// TIA Portal V18 program export: 5 tag tables, 0 data types, 1 data blocks, 15 code blocks (in call order from the OBs), 44 instance data blocks

VAR_GLOBAL   // PLC tag table "AI"
   "H/SSR_019_TT01_IN" AT %IW70 : Int;
   "H/SSR_019_TT02_IN" AT %IW72 : Int;
   "H/SSR_019_APT01_IN" AT %IW74 : Int;
   "H/SSR_019_GPT101_IN" AT %IW78 : Int;
   "H/SSR_019_GPT201_IN" AT %IW80 : Int;
   "H/SSR_019_GPT301_IN" AT %IW82 : Int;
   "H/SSR_019_GPT401_IN" AT %IW84 : Int;
   "H/SSR_019_GPT501_IN" AT %IW86 : Int;
   "H/SSR_019_GPT601_IN" AT %IW88 : Int;
   "H/SSR_019_TT03_IN" AT %IW76 : Int;
   Tag_1 AT %T5 : Timer;
END_VAR

VAR_GLOBAL   // PLC tag table "AO"
   "H/SSR_019_CV01_CVOUT" AT %QW26 : Int;
   "H/SSR_019_CV02_CVOUT" AT %QW28 : Int;
   "H/SSR_019_CV03_CVOUT" AT %QW30 : Int;
   SPARE AT %QW38 : Int;
   SPARE_1 AT %QW40 : Int;
   SPARE_2 AT %QW42 : Int;
   SPARE_3 AT %QW44 : Int;
   SPARE_4 AT %QW46 : Int;
   SPARE_5 AT %QW48 : Int;
   SPARE_6 AT %QW50 : Int;
   SPARE_7 AT %QW52 : Int;
   SPARE_8 AT %QW54 : Int;
   SPARE_9 AT %QW56 : Int;
   SPARE_10 AT %QW58 : Int;
   SPARE_11 AT %QW60 : Int;
   SPARE_12 AT %QW62 : Int;
   SPARE_13 AT %QW64 : Int;
   SPARE_14 AT %QW66 : Int;
END_VAR

VAR_GLOBAL   // PLC tag table "DI"
   "H/SSR_019_XV01_OPENFB" AT %I7.4 : Bool;
   "H/SSR_019_XV01_CLOSEFB" AT %I7.5 : Bool;
   "H/SSR_019_XV02_OPENFB" AT %I7.6 : Bool;
   "H/SSR_019_XV02_CLOSEFB" AT %I7.7 : Bool;
   "H/SSR_019_XV03_OPENFB" AT %I8.0 : Bool;
   "H/SSR_019_XV03_CLOSEFB" AT %I8.1 : Bool;
   "H/SSR_019_XV04_CLOSEFB" AT %I8.2 : Bool;
   "H/SSR_019_XV04_OPENFB" AT %I8.3 : Bool;
   "H/SSR_019_XV05_OPENFB" AT %I8.4 : Bool;
   "H/SSR_019_XV05_CLOSEFB" AT %I8.5 : Bool;
   "H/SSR_019_XV06_OPENFB" AT %I8.6 : Bool;
   "H/SSR_019_XV06_CLOSEFB" AT %I8.7 : Bool;
   "H/SSR_019_XV07_OPENFB" AT %I9.0 : Bool;
   "H/SSR_019_XV07_CLOSEFB" AT %I9.1 : Bool;
   "H/SSR_019_XV08_OPENFB" AT %I9.2 : Bool;
   "H/SSR_019_XV08_CLOSEFB" AT %I9.3 : Bool;
   "H/SSR_019_XV09_OPENFB" AT %I9.4 : Bool;
   "H/SSR_019_XV09_CLOSEFB" AT %I9.5 : Bool;
   "H/SSR_019_XV10_OPENFB" AT %I9.6 : Bool;
   "H/SSR_019_XV10_CLOSEFB" AT %I9.7 : Bool;
   "H/SSR_019_XV11_OPENFB" AT %I10.0 : Bool;
   "H/SSR_019_XV11_CLOSEFB" AT %I10.1 : Bool;
   "H/SSR_019_XV12_OPENFB" AT %I10.2 : Bool;
   "H/SSR_019_XV12_CLOSEFB" AT %I10.3 : Bool;
   "H/SSR_019_XV13_OPENFB" AT %I10.4 : Bool;
   "H/SSR_019_XV13_CLOSEFB" AT %I10.5 : Bool;
   "H/SSR_019_AG_RUNFB" AT %I10.6 : Bool;
   "H/SSR_019_AG_STOPFB" AT %I10.7 : Bool;
   "H/SSR_019_AG_TRIP" AT %I11.0 : Bool;
END_VAR

VAR_GLOBAL   // PLC tag table "DO"
   "H/SSR_006_XV01_OPEN" AT %Q0.0 : Bool;
   "H/SSR_006_XV02_OPEN" AT %Q0.1 : Bool;
   "H/SSR_006_XV03_OPEN" AT %Q0.2 : Bool;
   "H/SSR_006_XV04_OPEN" AT %Q0.3 : Bool;
   "H/SSR_006_XV05_OPEN" AT %Q0.4 : Bool;
   "H/SSR_006_XV06_OPEN" AT %Q0.5 : Bool;
   "H/SSR_006_XV07_OPEN" AT %Q0.6 : Bool;
   "H/SSR_006_XV08_OPEN" AT %Q0.7 : Bool;
   "H/SSR_006_XV09_OPEN" AT %Q1.0 : Bool;
   "H/SSR_006_XV10_OPEN" AT %Q1.1 : Bool;
   "H/SSR_006_XV11_OPEN" AT %Q1.2 : Bool;
   "H/SSR_006_XV12_OPEN" AT %Q1.3 : Bool;
   "H/SSR_006_XV13_OPEN" AT %Q1.4 : Bool;
   "H/SSR_006_XV14_OPEN" AT %Q1.5 : Bool;
   "H/SSR_006_AG_RUN" AT %Q1.6 : Bool;
   "H/SSR_010_XV01_OPEN" AT %Q1.7 : Bool;
   "H/SSR_010_XV02_OPEN" AT %Q2.0 : Bool;
   "H/SSR_010_XV03_OPEN" AT %Q2.1 : Bool;
   "H/SSR_010_XV04_OPEN" AT %Q2.2 : Bool;
   "H/SSR_010_XV05_OPEN" AT %Q2.3 : Bool;
   "H/SSR_010_XV06_OPEN" AT %Q2.4 : Bool;
   "H/SSR_010_XV07_OPEN" AT %Q2.5 : Bool;
   "H/SSR_010_XV08_OPEN" AT %Q2.6 : Bool;
   "H/SSR_010_XV09_OPEN" AT %Q2.7 : Bool;
   "H/SSR_010_XV10_OPEN" AT %Q3.0 : Bool;
   "H/SSR_010_XV11_OPEN" AT %Q3.1 : Bool;
   "H/SSR_010_XV12_OPEN" AT %Q3.2 : Bool;
   "H/SSR_010_XV13_OPEN" AT %Q3.3 : Bool;
   "H/SSR_010_XV14_OPEN" AT %Q3.4 : Bool;
   "H/SSR_010_AG_RUN" AT %Q3.5 : Bool;
   "H/SSR_019_XV01_OPEN" AT %Q3.6 : Bool;
   "H/SSR_019_XV02_OPEN" AT %Q3.7 : Bool;
   "H/SSR_019_XV03_OPEN" AT %Q4.0 : Bool;
   "H/SSR_019_XV04_OPEN" AT %Q4.1 : Bool;
   "H/SSR_019_XV05_OPEN" AT %Q4.2 : Bool;
   "H/SSR_019_XV06_OPEN" AT %Q4.3 : Bool;
   "H/SSR_019_XV07_OPEN" AT %Q4.4 : Bool;
   "H/SSR_019_XV08_OPEN" AT %Q4.5 : Bool;
   "H/SSR_019_XV09_OPEN" AT %Q4.6 : Bool;
   "H/SSR_019_XV10_OPEN" AT %Q4.7 : Bool;
   "H/SSR_019_XV11_OPEN" AT %Q5.0 : Bool;
   "H/SSR_019_XV12_OPEN" AT %Q5.1 : Bool;
   "H/SSR_019_XV13_OPEN" AT %Q5.2 : Bool;
   "H/SSR_019_XV14_OPEN" AT %Q5.3 : Bool;
   "H/SSR_019_AG_RUN" AT %Q5.4 : Bool;
   "H/SSR_020_XV01_OPEN" AT %Q5.5 : Bool;
   "H/SSR_020_XV02_OPEN" AT %Q5.6 : Bool;
   "H/SSR_020_XV03_OPEN" AT %Q5.7 : Bool;
   "H/SSR_020_XV04_OPEN" AT %Q6.0 : Bool;
   "H/SSR_020_XV05_OPEN" AT %Q6.1 : Bool;
   "H/SSR_020_XV06_OPEN" AT %Q6.2 : Bool;
   "H/SSR_020_XV07_OPEN" AT %Q6.3 : Bool;
   "H/SSR_020_XV08_OPEN" AT %Q6.4 : Bool;
   "H/SSR_020_XV09_OPEN" AT %Q6.5 : Bool;
   "H/SSR_020_XV10_OPEN" AT %Q6.6 : Bool;
   "H/SSR_020_XV11_OPEN" AT %Q6.7 : Bool;
   "H/SSR_020_XV12_OPEN" AT %Q7.0 : Bool;
   "H/SSR_020_XV13_OPEN" AT %Q7.1 : Bool;
   "H/SSR_020_XV14_OPEN" AT %Q7.2 : Bool;
   "H/SSR_020_AG_RUN" AT %Q7.3 : Bool;
   DO_SPARE_1 AT %Q7.4 : Bool;
   DO_SPARE_2 AT %Q7.5 : Bool;
   DO_SPARE_3 AT %Q7.6 : Bool;
   DO_SPARE_4 AT %Q7.7 : Bool;
   DO_SPARE_5 AT %Q8.0 : Bool;
   DO_SPARE_6 AT %Q8.1 : Bool;
   DO_SPARE_7 AT %Q8.2 : Bool;
   DO_SPARE_8 AT %Q8.3 : Bool;
   DO_SPARE_9 AT %Q8.4 : Bool;
   DO_SPARE_10 AT %Q8.5 : Bool;
   DO_SPARE_11 AT %Q8.6 : Bool;
   DO_SPARE_12 AT %Q8.7 : Bool;
   DO_SPARE_13 AT %Q9.0 : Bool;
   DO_SPARE_14 AT %Q9.1 : Bool;
   DO_SPARE_15 AT %Q9.2 : Bool;
   DO_SPARE_16 AT %Q9.3 : Bool;
   DO_SPARE_17 AT %Q9.4 : Bool;
   DO_SPARE_18 AT %Q9.5 : Bool;
   DO_SPARE_19 AT %Q9.6 : Bool;
   DO_SPARE_20 AT %Q9.7 : Bool;
   DO_SPARE_21 AT %Q10.0 : Bool;
   DO_SPARE_22 AT %Q10.1 : Bool;
   DO_SPARE_23 AT %Q10.2 : Bool;
   DO_SPARE_24 AT %Q10.3 : Bool;
   DO_SPARE_25 AT %Q10.4 : Bool;
   DO_SPARE_26 AT %Q10.5 : Bool;
   DO_SPARE_27 AT %Q10.6 : Bool;
   DO_SPARE_28 AT %Q10.7 : Bool;
   DO_SPARE_29 AT %Q11.0 : Bool;
   DO_SPARE_30 AT %Q11.1 : Bool;
   DO_SPARE_31 AT %Q11.2 : Bool;
   DO_SPARE_32 AT %Q11.3 : Bool;
   DO_SPARE_33 AT %Q11.4 : Bool;
   DO_SPARE_34 AT %Q11.5 : Bool;
   DO_SPARE_35 AT %Q11.6 : Bool;
   DO_SPARE_36 AT %Q11.7 : Bool;
   DO_SPARE_37 AT %Q12.0 : Bool;
   DO_SPARE_38 AT %Q12.1 : Bool;
   DO_SPARE_39 AT %Q12.2 : Bool;
   DO_SPARE_40 AT %Q12.3 : Bool;
   DO_SPARE_41 AT %Q12.4 : Bool;
   DO_SPARE_42 AT %Q12.5 : Bool;
   DO_SPARE_43 AT %Q12.6 : Bool;
   DO_SPARE_44 AT %Q12.7 : Bool;
   DO_SPARE_45 AT %Q13.0 : Bool;
   DO_SPARE_46 AT %Q13.1 : Bool;
   DO_SPARE_47 AT %Q13.2 : Bool;
   DO_SPARE_48 AT %Q13.3 : Bool;
   DO_SPARE_49 AT %Q13.4 : Bool;
   DO_SPARE_50 AT %Q13.5 : Bool;
   DO_SPARE_51 AT %Q13.6 : Bool;
   DO_SPARE_52 AT %Q13.7 : Bool;
END_VAR

VAR_GLOBAL   // PLC tag table "Default tag table_1"
   System_Byte AT %MB1 : Byte;
   FirstScan AT %M1.0 : Bool;
   DiagStatusUpdate AT %M1.1 : Bool;
   AlwaysTRUE AT %M1.2 : Bool;
   AlwaysFALSE AT %M1.3 : Bool;
   Clock_Byte AT %MB0 : Byte;
   Clock_10Hz AT %M0.0 : Bool;
   Clock_5Hz AT %M0.1 : Bool;
   "Clock_2.5Hz" AT %M0.2 : Bool;
   Clock_2Hz AT %M0.3 : Bool;
   "Clock_1.25Hz" AT %M0.4 : Bool;
   Clock_1Hz AT %M0.5 : Bool;
   "Clock_0.625Hz" AT %M0.6 : Bool;
   "Clock_0.5Hz" AT %M0.7 : Bool;
   "H/SSR_019_START" AT %M2.0 : Bool;
   "H/SSR_019_SP" AT %MD4 : Real;
   "H/SSR_019_TT01_PV" AT %MD8 : Real;
   "H/SSR_019_ALERT_SP" AT %MD12 : Real;
   "H/SSR_019_CHBr_RT_SP" AT %MD16 : Real;
   "H/SSR_019_RT_HW_SP" AT %MD20 : Real;
   "H/SSR_019_HW_STEAM_SP" AT %MD24 : Real;
   "H/SSR_019_RT_CHBr_SP" AT %MD28 : Real;
   "H/SSR_019_SOURCE_SEL" AT %MW32 : Int;
   "H/SSR_019_AM" AT %M2.1 : Bool;
   "H/SSR_019_TIME_SP" AT %MW34 : Int;
   "H/SSR_019_KP" AT %MW36 : Int;
   "H/SSR_019_TI" AT %MW38 : Int;
   "H/SSR_019_TT02_PV" AT %MD40 : Real;
   "H/SSR_019_CV02_MANOUT" AT %MD44 : Real;
   "H/SSR_019_START_PV" AT %MD48 : Real;
   "H/SSR_019_CV02_SCVOUT" AT %MD52 : Real;
   "H/SSR_019_RUN_MIN" AT %MW56 : Int;
   "H/SSR_019_FLUSH_TIME_SP" AT %MW60 : Int;
   "H/SSR_019_VENT_TIME_SP" AT %MW62 : Int;
   "H/SSR_019_CONDENSATE_TIME_SP" AT %MW64 : Int;
   "H/SSR_019_XV01_CMD" AT %M58.7 : Bool;
   "H/SSR_019_XV02_CMD" AT %M59.0 : Bool;
   "H/SSR_019_XV03_CMD" AT %M59.1 : Bool;
   "H/SSR_019_XV07_CMD" AT %M59.2 : Bool;
   "H/SSR_019_XV08_CMD" AT %M59.3 : Bool;
   "H/SSR_019_XV09_CMD" AT %M59.4 : Bool;
   "H/SSR_019_XV11_CMD" AT %M59.5 : Bool;
   "H/SSR_019_XV12_CMD" AT %M59.6 : Bool;
   "H/SSR_019_XV13_CMD" AT %M59.7 : Bool;
   "H/SSR_019_XV10_CMD" AT %M66.0 : Bool;
   "H/SSR_019_XV05_CMD" AT %M66.1 : Bool;
   "H/SSR_019_XV06_CMD" AT %M66.2 : Bool;
   "H/SSR_019_FLUSH_RUN_TIME" AT %MD68 : Real;
   "H/SSR_019_CONDENSATE_RUN_TIME" AT %MD72 : Real;
   "H/SSR_019_VENT_RUN_TIME" AT %MD76 : Real;
   "H/SSR_019_CV01_MANOUT" AT %MD80 : Real;
   "H/SSR_019_CV01_SCVOUT" AT %MD84 : Real;
   "H/SSR_019_HOLD" AT %M66.3 : Bool;
   "H/SSR_019_EMSTOP" AT %M66.4 : Bool;
   XV_ERRORMON_TIME AT %MD88 : Time;
   "H/SSR_019_XV01_RESET" AT %M66.5 : Bool;
   "H/SSR_019_XV01_MCMD" AT %M66.6 : Bool;
   "H/SSR_019_XV01_Status" AT %MW92 : Word;
   "H/SSR_019_XV02_MCMD" AT %M66.7 : Bool;
   "H/SSR_019_XV02_RESET" AT %M67.0 : Bool;
   "H/SSR_019_XV03_MCMD" AT %M67.1 : Bool;
   "H/SSR_019_XV03_RESET" AT %M67.2 : Bool;
   "H/SSR_019_XV04_MCMD" AT %M67.3 : Bool;
   "H/SSR_019_XV04_RESET" AT %M67.4 : Bool;
   "H/SSR_019_XV05_MCMD" AT %M67.5 : Bool;
   "H/SSR_019_XV05_RESET" AT %M67.6 : Bool;
   "H/SSR_019_XV06_MCMD" AT %M67.7 : Bool;
   "H/SSR_019_XV06_RESET" AT %M94.0 : Bool;
   "H/SSR_019_XV07_MCMD" AT %M94.1 : Bool;
   "H/SSR_019_XV07_RESET" AT %M94.2 : Bool;
   "H/SSR_019_XV08_MCMD" AT %M94.3 : Bool;
   "H/SSR_019_XV08_RESET" AT %M94.4 : Bool;
   "H/SSR_019_XV09_MCMD" AT %M94.5 : Bool;
   "H/SSR_019_XV09_RESET" AT %M94.6 : Bool;
   "H/SSR_019_XV10_MCMD" AT %M94.7 : Bool;
   "H/SSR_019_XV10_RESET" AT %M95.0 : Bool;
   "H/SSR_019_XV11_MCMD" AT %M95.1 : Bool;
   "H/SSR_019_XV11_RESET" AT %M95.2 : Bool;
   "H/SSR_019_XV12_MCMD" AT %M95.3 : Bool;
   "H/SSR_019_XV12_RESET" AT %M95.4 : Bool;
   "H/SSR_019_XV13_MCMD" AT %M95.5 : Bool;
   "H/SSR_019_XV13_RESET" AT %M95.6 : Bool;
   "H/SSR_019_XV02_Status" AT %MW96 : Word;
   "H/SSR_019_XV03_Status" AT %MW98 : Word;
   "H/SSR_019_XV04_Status" AT %MW100 : Word;
   "H/SSR_019_XV05_Status" AT %MW102 : Word;
   "H/SSR_019_XV07_Status" AT %MW104 : Word;
   "H/SSR_019_XV08_Status" AT %MW106 : Word;
   "H/SSR_019_XV09_Status" AT %MW108 : Word;
   "H/SSR_019_XV10_Status" AT %MW110 : Word;
   "H/SSR_019_XV06_Status" AT %MW112 : Word;
   "H/SSR_019_XV11_Status" AT %MW114 : Word;
   "H/SSR_019_XV12_Status" AT %MW116 : Word;
   "H/SSR_019_XV13_Status" AT %MW118 : Word;
   "H/SSR_019_CV03_SCVOUT" AT %MW120 : Int;
   "H/SSR_019_APT01_PV" AT %MD122 : Real;
   "H/SSR_019_AG_CMD" AT %M2.2 : Bool;
   "H/SSR_019_AG_MCMD" AT %M2.3 : Bool;
   "H/SSR_019_AG_RESET" AT %M2.4 : Bool;
   "H/SSR_019_AG_Status" AT %MW126 : Word;
   "H/SSR_019_CV03_MANOUT" AT %MD128 : Real;
   "H/SSR_019_TT01_Faulty" AT %M2.5 : Bool;
   "H/SSR_019_APT01_Faulty" AT %M2.6 : Bool;
   "H/SSR_019_TT02_Faulty" AT %M2.7 : Bool;
   "H/SSR_019_TT01_Fault" AT %M3.0 : Bool;
   "H/SSR_019_ALERT_SP_EMPTY" AT %M3.1 : Bool;
   "H/SSR_019_SP_EMPTY" AT %M3.2 : Bool;
   "H/SSR_019_CHANGEOVER_SP_EMPTY" AT %M3.3 : Bool;
   "H/SSR_019_FlushTime_SP_EMPTY" AT %M3.4 : Bool;
   "H/SSR_019_VentTime_SP_EMPTY" AT %M3.5 : Bool;
   "H/SSR_019_Cond_Time_EMPTY" AT %M3.6 : Bool;
   "H/SSR_019_XV01_Faulty" AT %M3.7 : Bool;
   "H/SSR_019_XV02_Faulty" AT %M58.0 : Bool;
   "H/SSR_019_XV03_Faulty" AT %M58.1 : Bool;
   "H/SSR_019_XV04_Faulty" AT %M58.2 : Bool;
   "H/SSR_019_XV05_Faulty" AT %M58.3 : Bool;
   "H/SSR_019_XV06_Faulty" AT %M58.4 : Bool;
   "H/SSR_019_XV07_Faulty" AT %M58.5 : Bool;
   "H/SSR_019_XV08_Faulty" AT %M58.6 : Bool;
   "H/SSR_019_XV09_Faulty" AT %M95.7 : Bool;
   "H/SSR_019_XV10_Faulty" AT %M132.0 : Bool;
   "H/SSR_019_XV11_Faulty" AT %M132.1 : Bool;
   "H/SSR_019_XV12_Faulty" AT %M132.2 : Bool;
   "H/SSR_019_XV13_Faulty" AT %M132.3 : Bool;
   "H/SSR_019_Flush_CMP" AT %M132.4 : Bool;
   "H/SSR_019_Vent_CMP" AT %M132.5 : Bool;
   "H/SSR_019_Cond_CMP" AT %M134.0 : Bool;
   "H/SSR_019_GPT101_Fault" AT %M134.1 : Bool;
   "H/SSR_019_GPT101_PV" AT %MD130 : Real;
   "H/SSR_019_GPT201_PV" AT %MD134 : Real;
   "H/SSR_019_GPT201_Fault" AT %M134.2 : Bool;
   "H/SSR_019_GPT301_Fault" AT %M134.3 : Bool;
   "H/SSR_019_GPT401_Fault" AT %M134.4 : Bool;
   "H/SSR_019_GPT501_Fault" AT %M134.5 : Bool;
   "H/SSR_019_GPT601_Fault" AT %M134.6 : Bool;
   "H/SSR_019_TT03_Fault" AT %M135.0 : Bool;
   "H/SSR_019_GPT301_PV" AT %MD132 : Real;
   "H/SSR_019_GPT401_PV" AT %MD135 : Real;
   "H/SSR_019_GPT501_PV" AT %MD136 : Real;
   "H/SSR_019_GPT601_PV" AT %MD137 : Real;
   "H/SSR_019_RESET" AT %M134.7 : Bool;
   "H/SSR_019_TT103_PV" AT %MD138 : Real;
   "H/SSR_019_HOOTER_Status" AT %M135.1 : Bool;
END_VAR
VAR_GLOBAL CONSTANT   // user constants
   "None(1)" : Pip := 65535;
   "Automatic update(1)" : Pip := 0;
   "PIP 1(1)" : Pip := 1;
   "PIP 2(1)" : Pip := 2;
   "PIP 3(1)" : Pip := 3;
   "PIP 4(1)" : Pip := 4;
   "PIP 5(1)" : Pip := 5;
   "PIP 6(1)" : Pip := 6;
   "PIP 7(1)" : Pip := 7;
   "PIP 8(1)" : Pip := 8;
   "PIP 9(1)" : Pip := 9;
   "PIP 10(1)" : Pip := 10;
   "PIP 11(1)" : Pip := 11;
   "PIP 12(1)" : Pip := 12;
   "PIP 13(1)" : Pip := 13;
   "PIP 14(1)" : Pip := 14;
   "PIP 15(1)" : Pip := 15;
   "PIP 16(1)" : Pip := 16;
   "PIP 17(1)" : Pip := 17;
   "PIP 18(1)" : Pip := 18;
   "PIP 19(1)" : Pip := 19;
   "PIP 20(1)" : Pip := 20;
   "PIP 21(1)" : Pip := 21;
   "PIP 22(1)" : Pip := 22;
   "PIP 23(1)" : Pip := 23;
   "PIP 24(1)" : Pip := 24;
   "PIP 25(1)" : Pip := 25;
   "PIP 26(1)" : Pip := 26;
   "PIP 27(1)" : Pip := 27;
   "PIP 28(1)" : Pip := 28;
   "PIP 29(1)" : Pip := 29;
   "PIP 30(1)" : Pip := 30;
   "PIP 31(1)" : Pip := 31;
   "Local1~MC" : Hw_SubModule := 65151;
   "Local1~Common" : Hw_SubModule := 65150;
   "Local1~Device" : Hw_Device := 65132;
   "Local1~Configuration" : Hw_SubModule := 65133;
   "Local1~RHSystem" : Hw_Device := 34;
   "Local1~Display" : Hw_SubModule := 65154;
   "Local1~Exec" : Hw_SubModule := 65152;
   Local1 : Hw_SubModule := 65149;
   "Local1~PROFINET_interface_1" : Hw_Interface := 65164;
   "Local1~PROFINET_interface_1~Port_1" : Hw_Interface := 65165;
   "Local1~PROFINET_interface_1~Port_2" : Hw_Interface := 65166;
   "Local1~PROFINET_interface_1~HsystemIPRef_1" : Hw_Interface := 257;
   "Local1~HCPUredCtrl" : Hw_SubModule := 65147;
   "Local2~MC" : Hw_SubModule := 65351;
   "Local2~Common" : Hw_SubModule := 65350;
   "Local2~Device" : Hw_Device := 65332;
   "Local2~Configuration" : Hw_SubModule := 65333;
   "Local2~Display" : Hw_SubModule := 65354;
   "Local2~Exec" : Hw_SubModule := 65352;
   Local2 : Hw_SubModule := 65349;
   "Local2~PROFINET_interface_1" : Hw_Interface := 65364;
   "Local2~PROFINET_interface_1~Port_1" : Hw_Interface := 65365;
   "Local2~PROFINET_interface_1~Port_2" : Hw_Interface := 65366;
   "Local2~PROFINET_interface_1~HsystemIPRef_1" : Hw_Interface := 268;
   "Local2~HCPUredCtrl" : Hw_SubModule := 65347;
   "OB_AutoLogic(1)" : OB_PCYCLE := 1;
   "OB_Main(1)" : OB_PCYCLE := 123;
   "OB_PID Cyclic interrupt(1)" : OB_Cyclic := 30;
   "OB_Cyclic interrupt(1)" : OB_Cyclic := 31;
END_VAR

DATA_BLOCK "SIM_VALVE"   // DB29
{ S7_Optimized_Access := 'FALSE' }
VERSION : 0.1
// stored: AutoNumber true, DBAccessibleFromOPCUA true, DBAccessibleFromWebserver true, IsOnlyStoredInLoadMemory false, IsWriteProtectedInAS false
   VAR
      "H/SSR_019_XV01_CLOSEFB" : Bool;
      "H/SSR_019_XV02_OPENFB" : Bool;
      "H/SSR_019_XV02_CLOSEFB" : Bool;
      "H/SSR_019_XV03_OPENFB" : Bool;
      "H/SSR_019_XV03_CLOSEFB" : Bool;
      "H/SSR_019_XV04_CLOSEFB" : Bool;
      "H/SSR_019_XV04_OPENFB" : Bool;
      "H/SSR_019_XV05_OPENFB" : Bool;
      "H/SSR_019_XV05_CLOSEFB" : Bool;
      "H/SSR_019_XV06_OPENFB" : Bool;
      "H/SSR_019_XV06_CLOSEFB" : Bool;
      "H/SSR_019_XV07_OPENFB" : Bool;
      "H/SSR_019_XV07_CLOSEFB" : Bool;
      "H/SSR_019_XV08_OPENFB" : Bool;
      "H/SSR_019_XV08_CLOSEFB" : Bool;
      "H/SSR_019_XV09_OPENFB" : Bool;
      "H/SSR_019_XV09_CLOSEFB" : Bool;
      "H/SSR_019_XV10_OPENFB" : Bool;
      "H/SSR_019_XV10_CLOSEFB" : Bool;
      "H/SSR_019_XV11_OPENFB" : Bool;
      "H/SSR_019_XV11_CLOSEFB" : Bool;
      "H/SSR_019_XV12_OPENFB" : Bool;
      "H/SSR_019_XV12_CLOSEFB" : Bool;
      "H/SSR_019_XV13_OPENFB" : Bool;
      "H/SSR_019_XV13_CLOSEFB" : Bool;
      "H/SSR_019_TT01_IN" : Int;
      "H/SSR_019_TT02_IN" : Int;
      "H/SSR_019_APT01_IN" : Int;
      "H/SSR_019_GPT101_IN" : Int;
      "H/SSR_019_GPT201_IN" : Int;
      "H/SSR_019_GPT301_IN" : Int;
      "H/SSR_019_GPT401_IN" : Int;
      "H/SSR_019_GPT501_IN" : Int;
      "H/SSR_019_GPT601_IN" : Int;
      "H/SSR_019_TT03_IN" : Int;
      "H/SSR_019_TT01_PV" : Int;
      "H/SSR_019_XV01_OPENFB" : Bool;
      "H/SSR_019_TT02_INpv" : Bool;
      "H/SSR_019_APT01_PV" : Bool;
      "H/SSR_019_GPT101_PV" : Bool;
      "H/SSR_019_GPT201_PV" : Bool;
      "H/SSR_019_GPT301_PV" : Bool;
      "H/SSR_019_GPT401_PV" : Bool;
      "H/SSR_019_GPT501_PV" : Bool;
      "H/SSR_019_GPT601_PV" : Bool;
      "H/SSR_019_TT03_PV" : Bool;
      "H/SSR_019_TT01_PV_1" : Bool;
   END_VAR
BEGIN
END_DATA_BLOCK

ORGANIZATION_BLOCK "AutoLogic"   // OB1, FBD, ProgramCycle
TITLE = "Main Program Sweep (Cycle)"
{ S7_Optimized_Access := 'TRUE' }
VERSION : 0.1
// stored: AutoNumber true, IsIECCheckEnabled false, SetENOAutomatically false
   VAR_INPUT
      Initial_Call : Bool;   // Initial call of this OB
      Remanence : Bool;   // =True, if remanent data are available
   END_VAR
   VAR_TEMP
      UTL_TIME : Array[0..2] of DInt;
      chbs_cmd : Bool;
      chbr_cmd : Bool;
      STEAM_MAN_SCV_MVE : Real;
      STEAM_SCV_MVE : Real;
      STEAM_SCV_SCL : Real;
   END_VAR
BEGIN

REGION Network 1: Source select
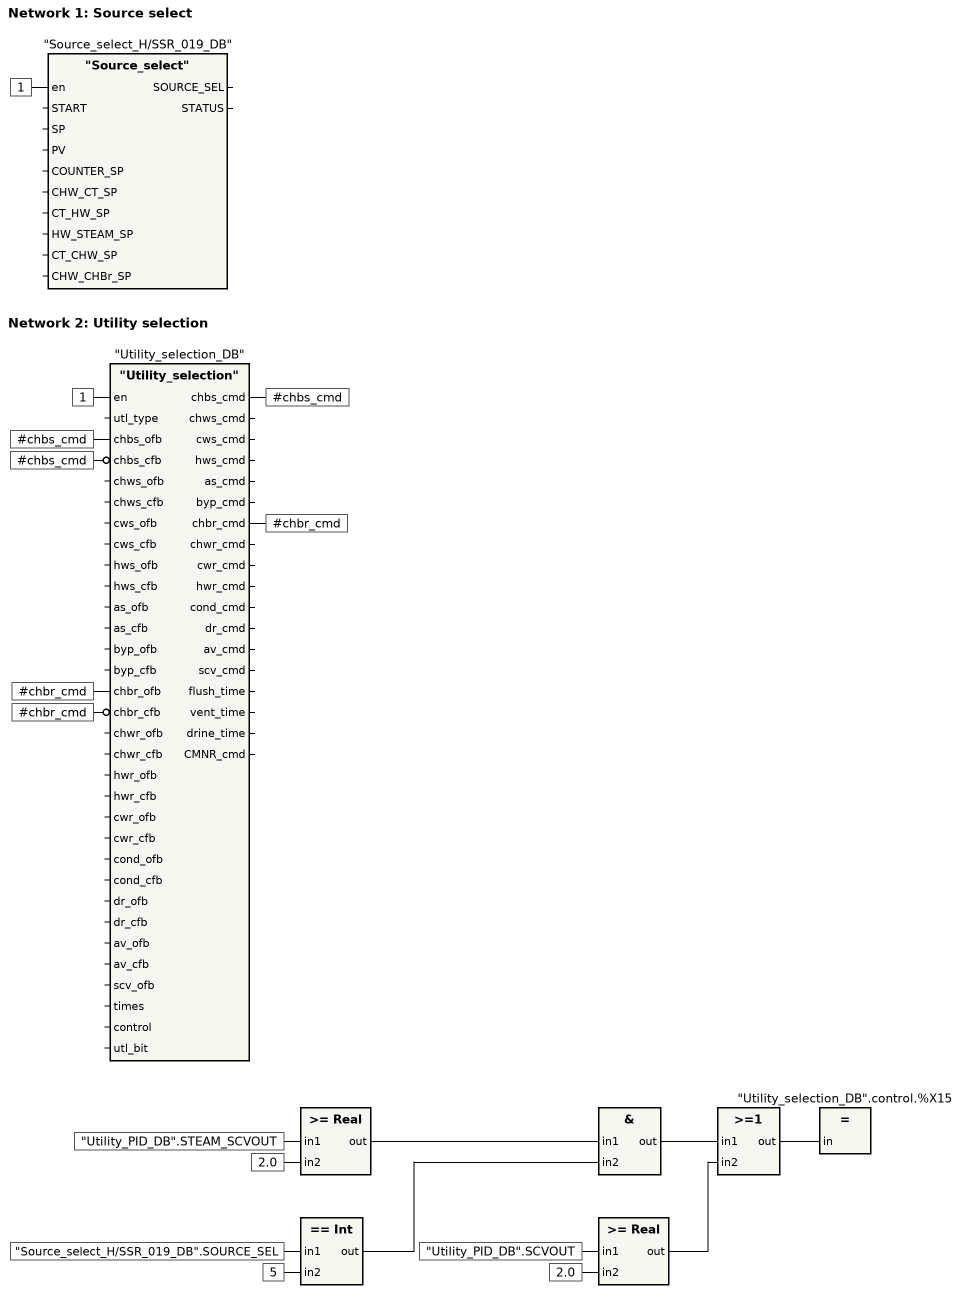
   IF 1 THEN
       "Source_select_H/SSR_019_DB"();   // "Source_select"
   END_IF;
END_REGION

REGION Network 2: Utility selection
   IF 1 THEN
       "Utility_selection_DB"(chbs_ofb := #chbs_cmd,   // "Utility_selection"
                              chbs_cfb := NOT #chbs_cmd,
                              chbr_ofb := #chbr_cmd,
                              chbr_cfb := NOT #chbr_cmd,
                              chbs_cmd => #chbs_cmd,
                              chbr_cmd => #chbr_cmd);
   END_IF;
   "Utility_selection_DB".control.%X15 := (("Utility_PID_DB".STEAM_SCVOUT >= 2.0) AND ("Source_select_H/SSR_019_DB".SOURCE_SEL = 5)) OR ("Utility_PID_DB".SCVOUT >= 2.0);
END_REGION
END_ORGANIZATION_BLOCK

FUNCTION_BLOCK "Source_select"   // FB1, FBD
TITLE = Source selection
{ S7_Optimized_Access := 'TRUE' }
VERSION : 0.1
// Source select
// stored: AutoNumber true, IsIECCheckEnabled false, IsRetainMemResEnabled false, MemoryReserve 100, SetENOAutomatically false, UDAEnableTagReadback false
   VAR_INPUT
      START : Bool;
      SP : Real;
      PV : Real;
      COUNTER_SP : Real;
      CHW_CT_SP : Real;
      CT_HW_SP : Real;
      HW_STEAM_SP : Real;
      CT_CHW_SP : Real;
      CHW_CHBr_SP : Real;
   END_VAR
   VAR_OUTPUT
      SOURCE_SEL : Int;
      STATUS : Word;
   END_VAR
   VAR
      Heating : Int;
      Cooling : Int;
      SUB_SP_COUNTER_SP : Real;
      ADD_SP_COUNTER_SP : Real;
      SS_TP1 { S7_SetPoint := 'True'} : TP_TIME;
      SS_TP2 { S7_SetPoint := 'True'} : TP_TIME;
      SS_TP3 { S7_SetPoint := 'True'} : TP_TIME;
      SS_TP4 { S7_SetPoint := 'True'} : TP_TIME;
      SS_TP5 { S7_SetPoint := 'True'} : TP_TIME;
      SS_TP6 { S7_SetPoint := 'True'} : TP_TIME;
      SS_TON1 { S7_SetPoint := 'True'} : TON_TIME;
      SS_TON3 { S7_SetPoint := 'True'} : TON_TIME;
      SS_TON4 { S7_SetPoint := 'True'} : TON_TIME;
      SS_TON5 { S7_SetPoint := 'True'} : TON_TIME;
      SS_TON6 { S7_SetPoint := 'True'} : TON_TIME;
      SS_TON7 { S7_SetPoint := 'True'} : TON_TIME;
   END_VAR
BEGIN

REGION Network 1: Heating
   // Heating
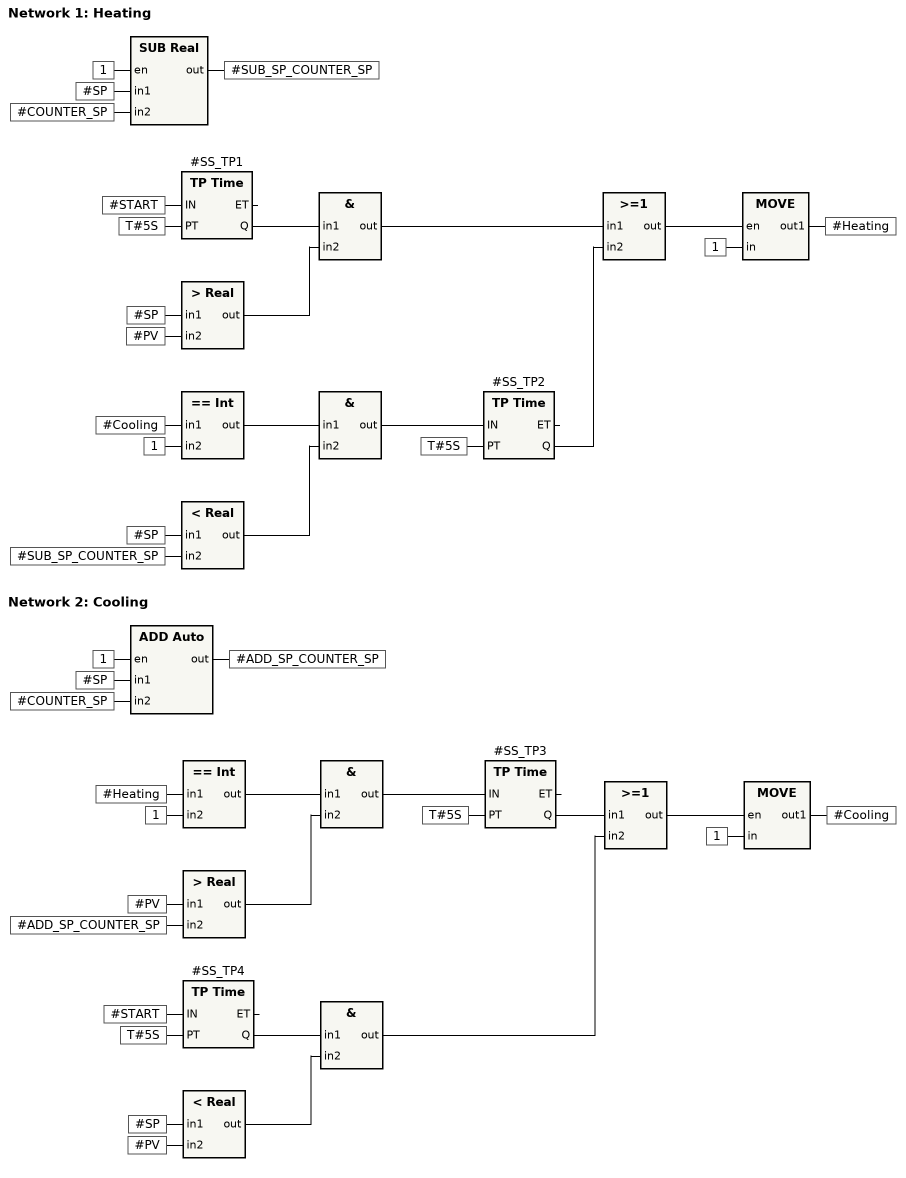
   IF 1 THEN #SUB_SP_COUNTER_SP := #SP - #COUNTER_SP; END_IF;
   #SS_TP1(IN := #START, PT := T#5S);   // TP
   #SS_TP2(IN := (#Cooling = 1) AND (#SP < #SUB_SP_COUNTER_SP), PT := T#5S);   // TP
   IF (#SS_TP1.Q AND (#SP > #PV)) OR #SS_TP2.Q THEN #Heating := 1; END_IF;
END_REGION

REGION Network 2: Cooling
   // Cooling
   IF 1 THEN #ADD_SP_COUNTER_SP := #SP + #COUNTER_SP; END_IF;
   #SS_TP3(IN := (#Heating = 1) AND (#PV > #ADD_SP_COUNTER_SP), PT := T#5S);   // TP
   #SS_TP4(IN := #START, PT := T#5S);   // TP
   IF #SS_TP3.Q OR (#SS_TP4.Q AND (#SP < #PV)) THEN #Cooling := 1; END_IF;
END_REGION

REGION Network 3: Heating & Cooling Reset
   // Heating & Cooling Reset
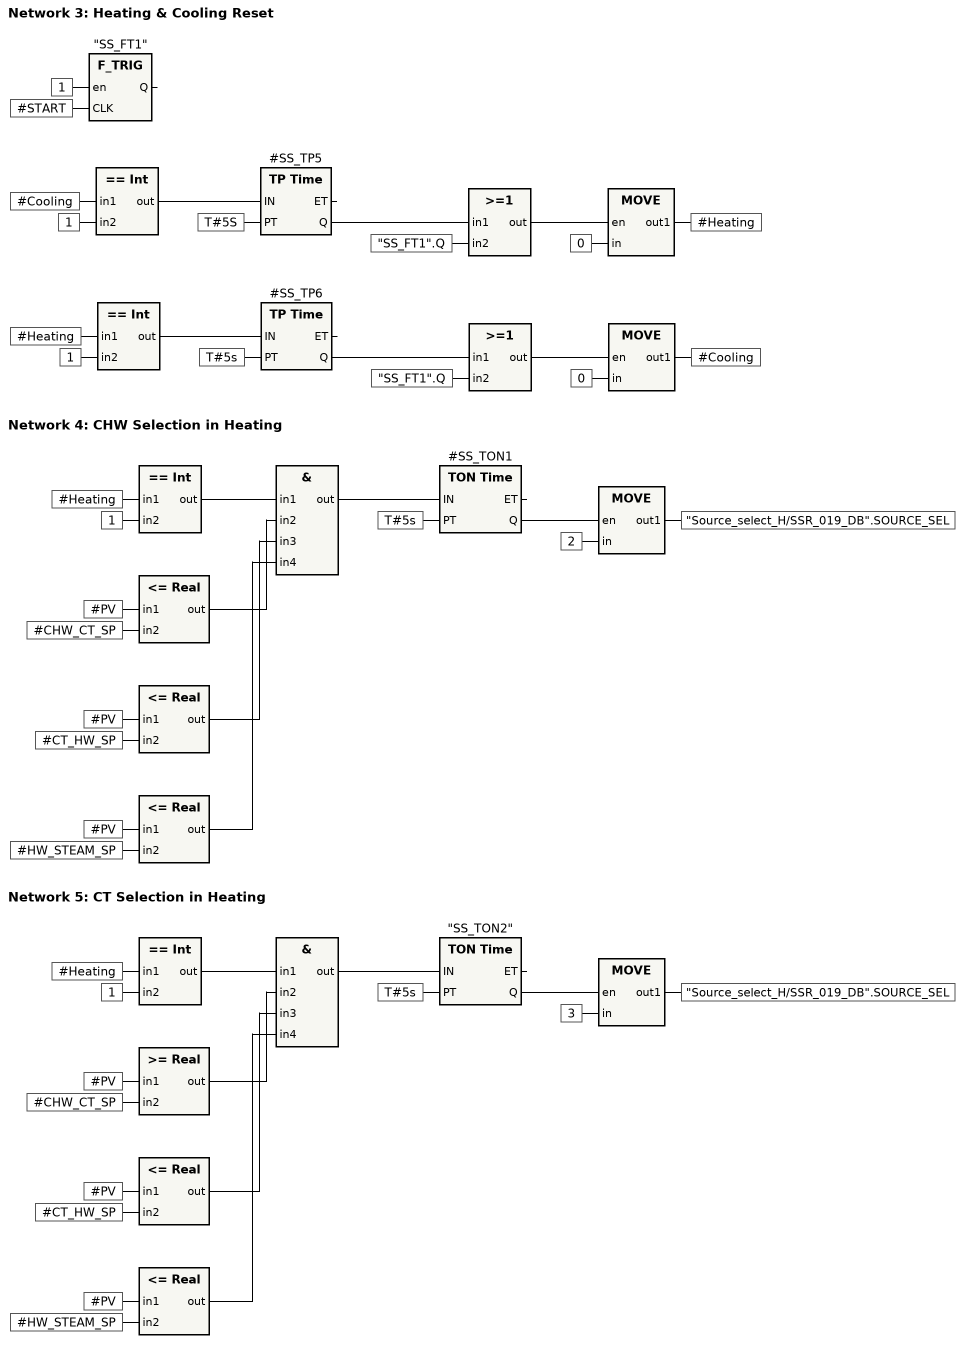
   IF 1 THEN
       "SS_FT1"(CLK := #START);   // F_TRIG
   END_IF;
   #SS_TP5(IN := #Cooling = 1, PT := T#5S);   // TP
   IF #SS_TP5.Q OR "SS_FT1".Q THEN #Heating := 0; END_IF;
   #SS_TP6(IN := #Heating = 1, PT := T#5s);   // TP
   IF #SS_TP6.Q OR "SS_FT1".Q THEN #Cooling := 0; END_IF;
END_REGION

REGION Network 4: CHW Selection in Heating
   // CHW Selection in Heating
   #SS_TON1(IN := (#Heating = 1) AND (#PV <= #CHW_CT_SP) AND (#PV <= #CT_HW_SP) AND (#PV <= #HW_STEAM_SP),   // TON
            PT := T#5s);
   IF #SS_TON1.Q THEN "Source_select_H/SSR_019_DB".SOURCE_SEL := 2; END_IF;
END_REGION

REGION Network 5: CT Selection in Heating
   // CT Selection in Heating
   "SS_TON2".TON(IN := (#Heating = 1) AND (#PV >= #CHW_CT_SP) AND (#PV <= #CT_HW_SP) AND (#PV <= #HW_STEAM_SP),
                 PT := T#5s);
   IF "SS_TON2".Q THEN "Source_select_H/SSR_019_DB".SOURCE_SEL := 3; END_IF;
END_REGION

REGION Network 6: HW Selection in Heating
   // HW Selection in Heating
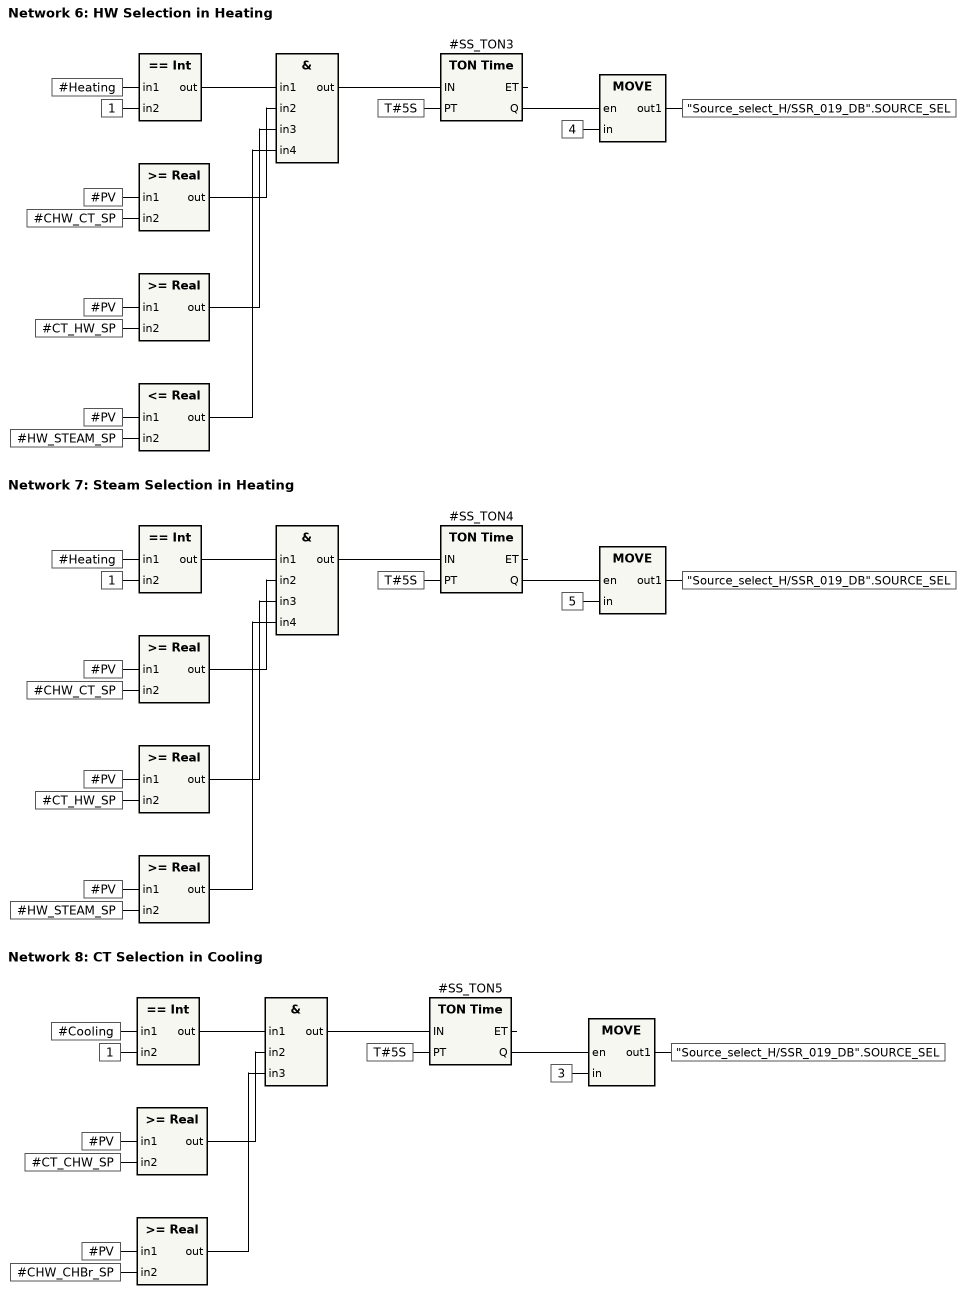
   #SS_TON3(IN := (#Heating = 1) AND (#PV >= #CHW_CT_SP) AND (#PV >= #CT_HW_SP) AND (#PV <= #HW_STEAM_SP),   // TON
            PT := T#5S);
   IF #SS_TON3.Q THEN "Source_select_H/SSR_019_DB".SOURCE_SEL := 4; END_IF;
END_REGION

REGION Network 7: Steam Selection in Heating
   // Steam Selection in Heating
   #SS_TON4(IN := (#Heating = 1) AND (#PV >= #CHW_CT_SP) AND (#PV >= #CT_HW_SP) AND (#PV >= #HW_STEAM_SP),   // TON
            PT := T#5S);
   IF #SS_TON4.Q THEN "Source_select_H/SSR_019_DB".SOURCE_SEL := 5; END_IF;
END_REGION

REGION Network 8: CT Selection in Cooling
   // CT Selection in Cooling
   #SS_TON5(IN := (#Cooling = 1) AND (#PV >= #CT_CHW_SP) AND (#PV >= #CHW_CHBr_SP), PT := T#5S);   // TON
   IF #SS_TON5.Q THEN "Source_select_H/SSR_019_DB".SOURCE_SEL := 3; END_IF;
END_REGION

REGION Network 9: CHW Selection in Cooling
   // CHW Selection in Cooling
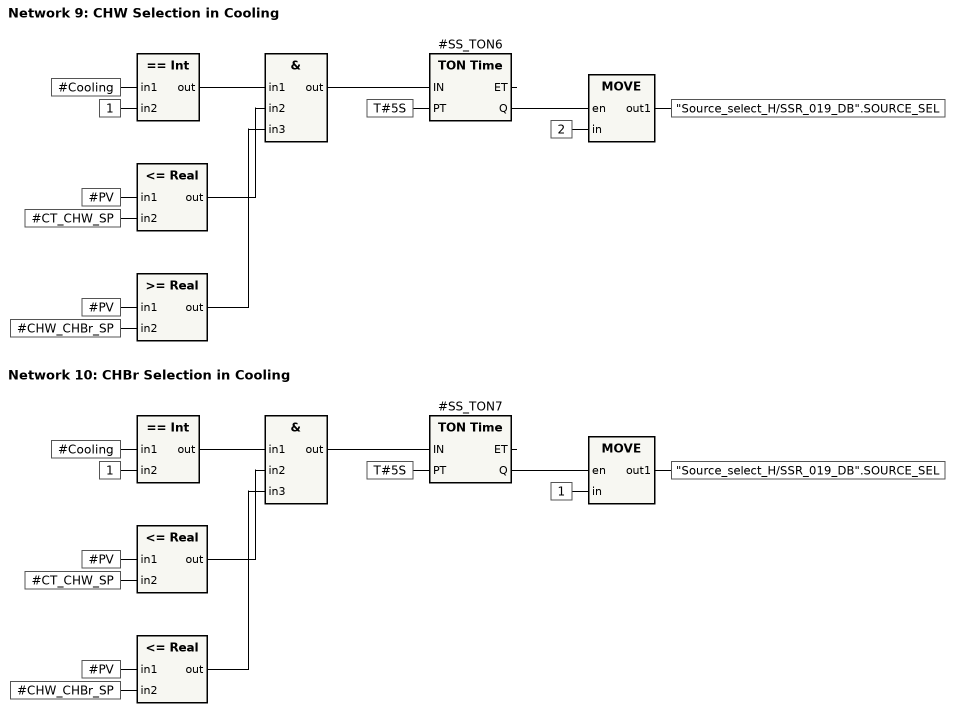
   #SS_TON6(IN := (#Cooling = 1) AND (#PV <= #CT_CHW_SP) AND (#PV >= #CHW_CHBr_SP), PT := T#5S);   // TON
   IF #SS_TON6.Q THEN "Source_select_H/SSR_019_DB".SOURCE_SEL := 2; END_IF;
END_REGION

REGION Network 10: CHBr Selection in Cooling
   // CHBr Selection in Cooling
   #SS_TON7(IN := (#Cooling = 1) AND (#PV <= #CT_CHW_SP) AND (#PV <= #CHW_CHBr_SP), PT := T#5S);   // TON
   IF #SS_TON7.Q THEN "Source_select_H/SSR_019_DB".SOURCE_SEL := 1; END_IF;
END_REGION
END_FUNCTION_BLOCK

FUNCTION_BLOCK "Utility_selection"   // FB7, FBD
TITLE = Selection1_12 , flushing13
{ S7_Optimized_Access := 'TRUE' }
VERSION : 0.1
// stored: AutoNumber false, IsIECCheckEnabled false, IsRetainMemResEnabled false, MemoryReserve 100, SetENOAutomatically false, UDAEnableTagReadback false
   VAR_INPUT
      utl_type : Int;
      chbs_ofb : Bool;
      chbs_cfb : Bool;
      chws_ofb : Bool;
      chws_cfb : Bool;
      cws_ofb : Bool;
      cws_cfb : Bool;
      hws_ofb : Bool;
      hws_cfb : Bool;
      as_ofb : Bool;
      as_cfb : Bool;
      byp_ofb : Bool;
      byp_cfb : Bool;
      chbr_ofb : Bool;
      chbr_cfb : Bool;
      chwr_ofb : Bool;
      chwr_cfb : Bool;
      hwr_ofb : Bool;
      hwr_cfb : Bool;
      cwr_ofb : Bool;
      cwr_cfb : Bool;
      cond_ofb : Bool;
      cond_cfb : Bool;
      dr_ofb : Bool;
      dr_cfb : Bool;
      av_ofb : Bool;
      av_cfb : Bool;
      scv_ofb : Bool;
      times : Array[0..2] of DInt;
   END_VAR
   VAR_OUTPUT
      chbs_cmd : Bool;
      chws_cmd : Bool;
      cws_cmd : Bool;
      hws_cmd : Bool;
      as_cmd : Bool;
      byp_cmd : Bool;
      chbr_cmd : Bool;
      chwr_cmd : Bool;
      cwr_cmd : Bool;
      hwr_cmd : Bool;
      cond_cmd : Bool;
      dr_cmd : Bool;
      av_cmd : Bool;
      scv_cmd : Bool;
      flush_time : DInt;
      vent_time : DInt;
      drine_time : DInt;
      CMNR_cmd : Bool;
   END_VAR
   VAR_IN_OUT
      control { ExternalVisible := 'False'} : Word;
      utl_bit : Bool;
   END_VAR
   VAR
      selection : Int;
      br_sel : Bool;
      chw_sel : Bool;
      cw_sel : Bool;
      hw_sel : Bool;
      flush_sel : Bool;
      st_sel : Bool;
      prev_util : Int;
      vent_start : Bool;
      start_temp : Bool;
      start : Bool;
      flush_tm_comp : Bool;
      am : Bool;
      pause : Bool;
      chbr_cmd1 : Bool;
      chbr_cmd2 : Bool;
      agr_fail : Bool;
      hold : Bool;
      hold_t : Bool;
      status : Word;
      steam_flush : Bool;
      SUV_flush : Bool;
      Pres_low : Bool;
      uti_cv : Bool;
      hw_autoflush : Bool;
      emstop : Bool;
      temp : Bool;
      en_flush : Bool;
      dr_start : Bool;
      hwr_cmd1 : Bool;
      hwr_cmd2 : Bool;
      chwr_cmd1 : Bool;
      chwr_cmd2 : Bool;
      cond_cmd1 : Bool;
      cwr_cmd1 : Bool;
      cwr_cmd2 : Bool;
      br_flush : Bool;
      chw_flush : Bool;
      cw_flush : Bool;
      hw_flush : Bool;
      st_flush : Bool;
      byp_cmd2 : Bool;
      Flush_Dint : DInt;
      Flush_Ptime : Time;
      Flush_Etime : Time;
      Flush_TTime : DInt;
      Vent_Etime : Time;
      Vent_TTime : DInt;
      Vent_Ptime : Time;
      Vent_Dint : DInt;
      Cond_Dint : DInt;
      Cond_Ptime : Time;
      Cond_Etime : Time;
      Cond_TTime : DInt;
      reserved : Bool;
      Vent_tm_comp : Bool;
      Cond_tm_comp : Bool;
      US_TOF3 { S7_SetPoint := 'True'} : TOF_TIME;
      US_TON2 { S7_SetPoint := 'True'} : TON_TIME;
      US_TON3 { S7_SetPoint := 'True'} : TON_TIME;
      US_TON4 { S7_SetPoint := 'True'} : TON_TIME;
      US_TON5 { S7_SetPoint := 'True'} : TON_TIME;
      US_TP2 { S7_SetPoint := 'True'} : TP_TIME;
      US_TP3 { S7_SetPoint := 'True'} : TP_TIME;
      US_TP4 { S7_SetPoint := 'True'} : TP_TIME;
      US_TOF1 { S7_SetPoint := 'True'} : TOF_TIME;
      UP_TP6 { S7_SetPoint := 'True'} : TP_TIME;
      US_TP8 { S7_SetPoint := 'True'} : TP_TIME;
      US_TP7 { S7_SetPoint := 'True'} : TP_TIME;
      US_TP9 { S7_SetPoint := 'True'} : TP_TIME;
      UP_TP1 { S7_SetPoint := 'True'} : TP_TIME;
      US_TP10 { S7_SetPoint := 'True'} : TP_TIME;
      US_TOF2 { S7_SetPoint := 'True'} : TOF_TIME;
      US_TOF4 { S7_SetPoint := 'True'} : TOF_TIME;
      US_TOF6 { S7_SetPoint := 'True'} : TOF_TIME;
      US_TP11 { S7_SetPoint := 'True'} : TP_TIME;
      US_TP12 { S7_SetPoint := 'True'} : TP_TIME;
      US_TON6 { S7_SetPoint := 'True'} : TON_TIME;
      US_TP5 { S7_SetPoint := 'True'} : TP_TIME;
      US_TON7 { S7_SetPoint := 'True'} : TON_TIME;
      US_TP13 { S7_SetPoint := 'True'} : TP_TIME;
      US_TP14 { S7_SetPoint := 'True'} : TP_TIME;
      US_TON8 { S7_SetPoint := 'True'} : TON_TIME;
      US_TP15 { S7_SetPoint := 'True'} : TP_TIME;
      US_TP20 { S7_SetPoint := 'True'} : TP_TIME;
      US_TON10 { S7_SetPoint := 'True'} : TON_TIME;
      US_TP16 { S7_SetPoint := 'True'} : TP_TIME;
      US_TON9 { S7_SetPoint := 'True'} : TON_TIME;
      US_TP17 { S7_SetPoint := 'True'} : TP_TIME;
      US_TP21 { S7_SetPoint := 'True'} : TP_TIME;
      S_TON11 { S7_SetPoint := 'True'} : TON_TIME;
      US_TP18 { S7_SetPoint := 'True'} : TP_TIME;
      US_TP19 { S7_SetPoint := 'True'} : TP_TIME;
   END_VAR
   VAR_TEMP   // added for the SCL form of the ladder/FBD networks
      _w1 : Bool;
   END_VAR
BEGIN

REGION Network 1: utility selection and moving
   // utility selection and moving
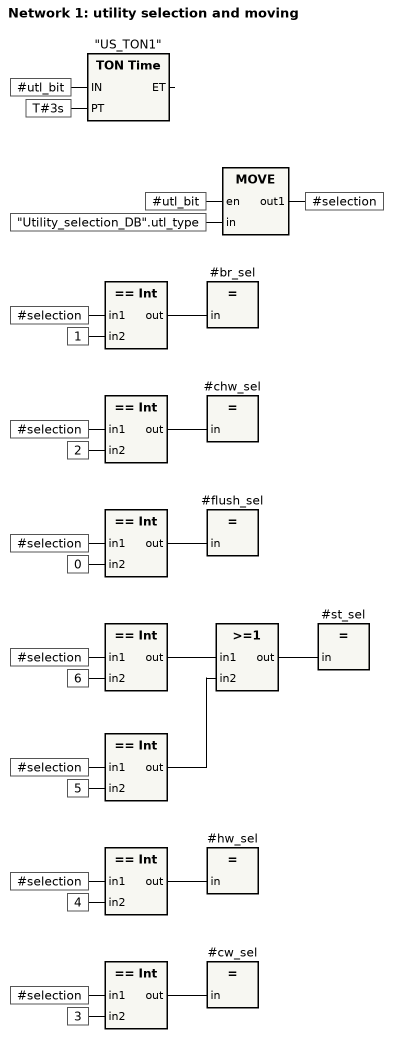
   "US_TON1".TON(IN := #utl_bit, PT := T#3s);
   IF #utl_bit THEN #selection := "Utility_selection_DB".utl_type; END_IF;
   #br_sel := #selection = 1;
   #chw_sel := #selection = 2;
   #flush_sel := #selection = 0;
   #st_sel := (#selection = 6) OR (#selection = 5);
   #hw_sel := #selection = 4;
   #cw_sel := #selection = 3;
END_REGION

REGION Network 2: previous utiliy identifucation
   // previous utiliy identifucation
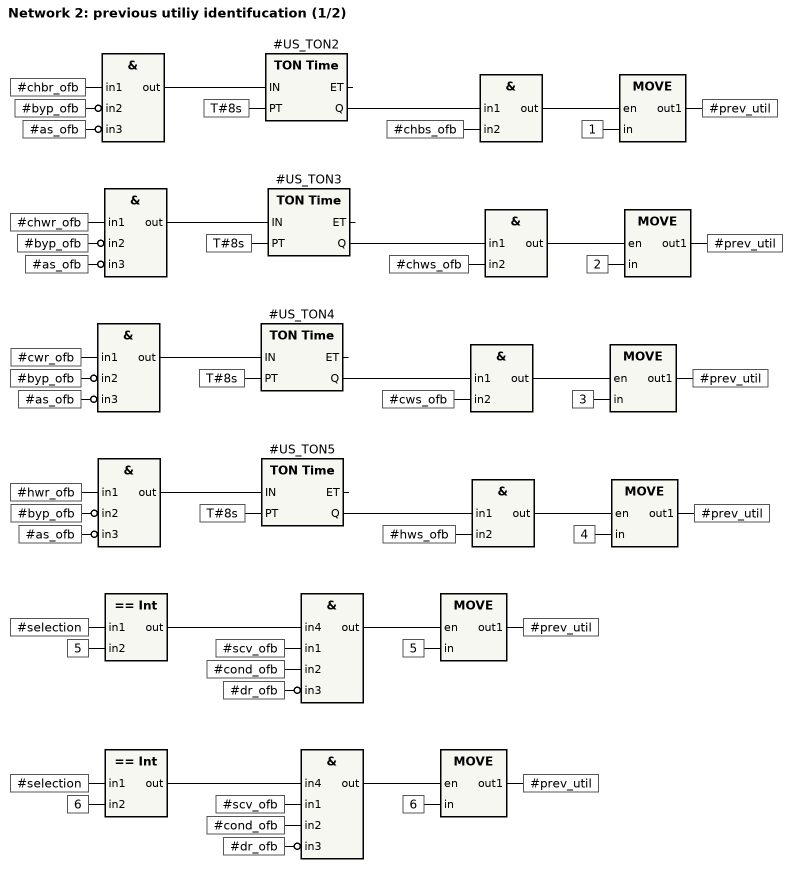
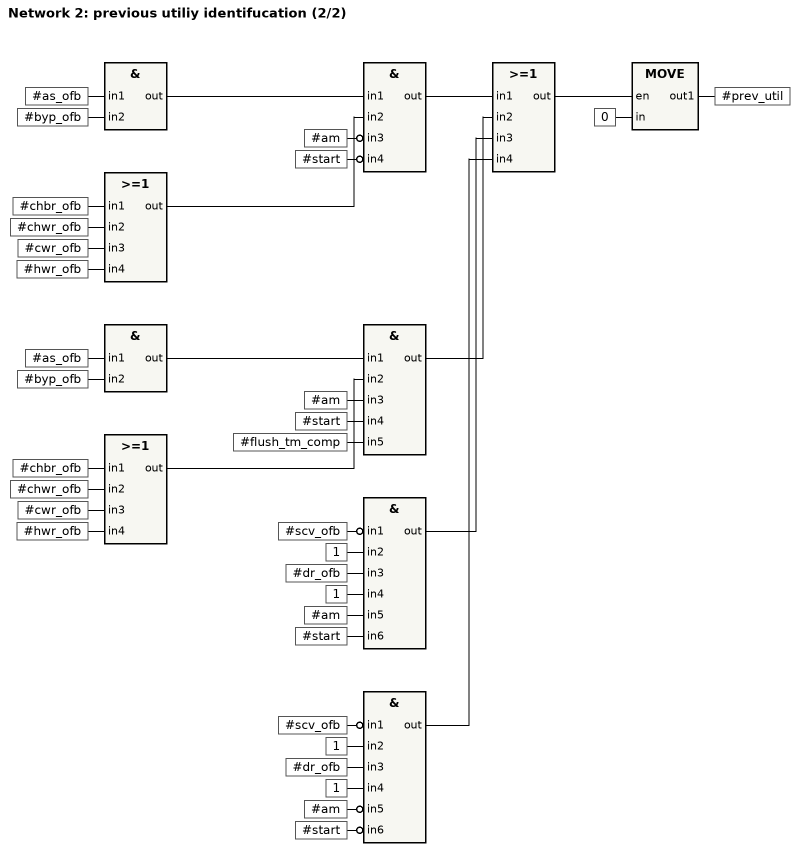
   #US_TON2(IN := #chbr_ofb AND NOT #byp_ofb AND NOT #as_ofb, PT := T#8s);   // TON
   IF #US_TON2.Q AND #chbs_ofb THEN #prev_util := 1; END_IF;
   #US_TON3(IN := #chwr_ofb AND NOT #byp_ofb AND NOT #as_ofb, PT := T#8s);   // TON
   IF #US_TON3.Q AND #chws_ofb THEN #prev_util := 2; END_IF;
   #US_TON4(IN := #cwr_ofb AND NOT #byp_ofb AND NOT #as_ofb, PT := T#8s);   // TON
   IF #US_TON4.Q AND #cws_ofb THEN #prev_util := 3; END_IF;
   #US_TON5(IN := #hwr_ofb AND NOT #byp_ofb AND NOT #as_ofb, PT := T#8s);   // TON
   IF #US_TON5.Q AND #hws_ofb THEN #prev_util := 4; END_IF;
   IF (#selection = 5) AND #scv_ofb AND #cond_ofb AND NOT #dr_ofb THEN #prev_util := 5; END_IF;
   IF (#selection = 6) AND #scv_ofb AND #cond_ofb AND NOT #dr_ofb THEN #prev_util := 6; END_IF;
   IF (#as_ofb AND #byp_ofb AND (#chbr_ofb OR #chwr_ofb OR #cwr_ofb OR #hwr_ofb) AND NOT #am AND NOT #start) OR (#as_ofb AND #byp_ofb AND (#chbr_ofb OR #chwr_ofb OR #cwr_ofb OR #hwr_ofb) AND #am AND #start AND #flush_tm_comp) OR (NOT #scv_ofb AND 1 AND #dr_ofb AND 1 AND #am AND #start) OR (NOT #scv_ofb AND 1 AND #dr_ofb AND 1 AND NOT #am AND NOT #start) THEN
       #prev_util := 0;
   END_IF;
END_REGION

REGION Network 3: flushing Identification
   // flushing Identification
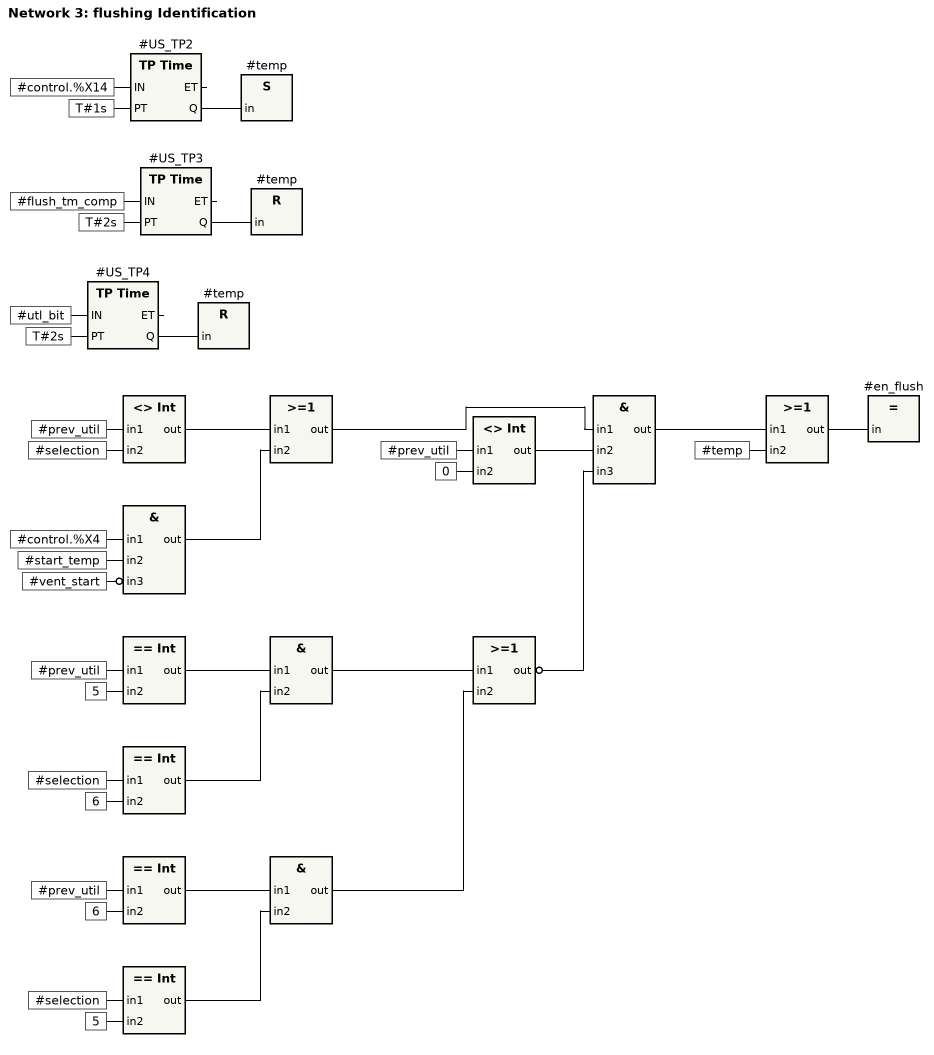
   #US_TP2(IN := #control.%X14, PT := T#1s);   // TP
   IF #US_TP2.Q THEN #temp := TRUE; END_IF;
   #US_TP3(IN := #flush_tm_comp, PT := T#2s);   // TP
   IF #US_TP3.Q THEN #temp := FALSE; END_IF;
   #US_TP4(IN := #utl_bit, PT := T#2s);   // TP
   IF #US_TP4.Q THEN #temp := FALSE; END_IF;
   #en_flush := (((#prev_util <> #selection) OR (#control.%X4 AND #start_temp AND NOT #vent_start)) AND (#prev_util <> 0) AND NOT (((#prev_util = 5) AND (#selection = 6)) OR ((#prev_util = 6) AND (#selection = 5)))) OR #temp;
END_REGION

REGION Network 4: temp_start
   // temp_start
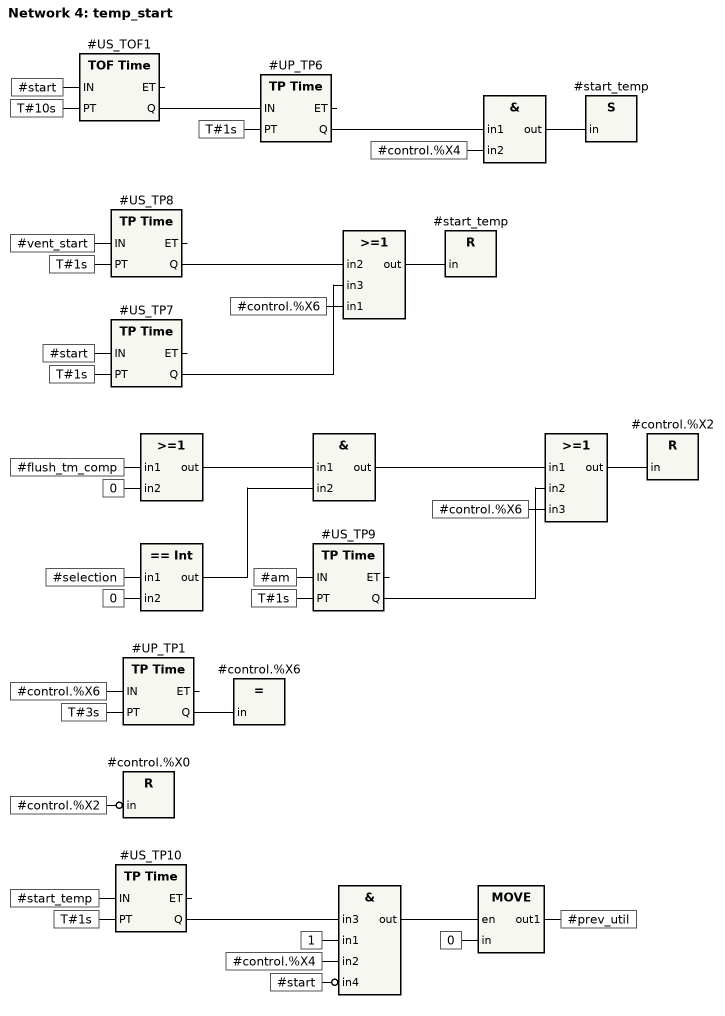
   #US_TOF1(IN := #start, PT := T#10s);   // TOF
   #UP_TP6(IN := #US_TOF1.Q, PT := T#1s);   // TP
   IF #UP_TP6.Q AND #control.%X4 THEN #start_temp := TRUE; END_IF;
   #US_TP8(IN := #vent_start, PT := T#1s);   // TP
   #US_TP7(IN := #start, PT := T#1s);   // TP
   IF #US_TP8.Q OR #US_TP7.Q OR #control.%X6 THEN #start_temp := FALSE; END_IF;
   #US_TP9(IN := #am, PT := T#1s);   // TP
   IF ((#flush_tm_comp OR 0) AND (#selection = 0)) OR #US_TP9.Q OR #control.%X6 THEN
       #control.%X2 := FALSE;
   END_IF;
   #UP_TP1(IN := #control.%X6, PT := T#3s);   // TP
   #control.%X6 := #UP_TP1.Q;
   IF NOT #control.%X2 THEN #control.%X0 := FALSE; END_IF;
   #US_TP10(IN := #start_temp, PT := T#1s);   // TP
   IF #US_TP10.Q AND 1 AND #control.%X4 AND NOT #start THEN #prev_util := 0; END_IF;
END_REGION

REGION Network 5: control and status word
   // control and status word
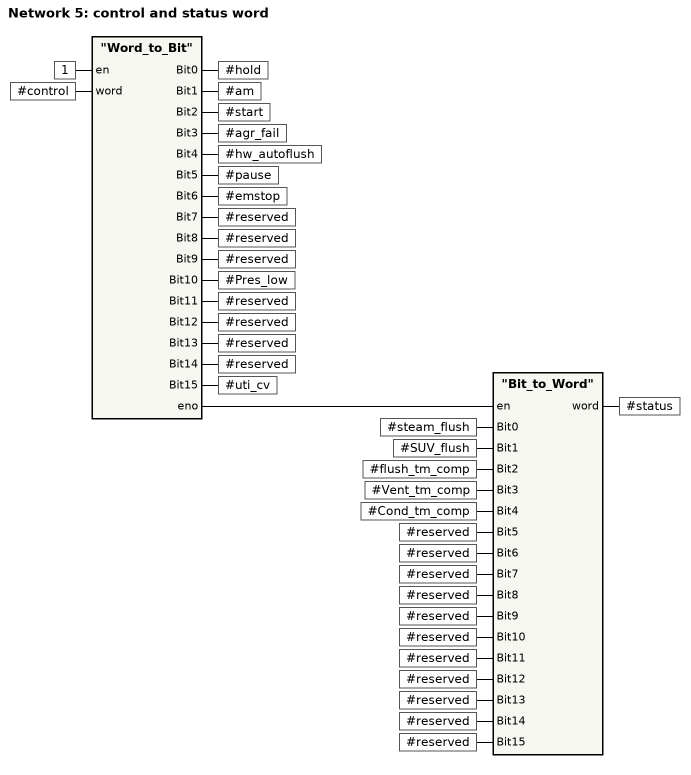
   "Word_to_Bit"(EN := 1,
                 "word" := #control,
                 Bit0 => #hold,
                 Bit1 => #am,
                 Bit2 => #start,
                 Bit3 => #agr_fail,
                 Bit4 => #hw_autoflush,
                 Bit5 => #pause,
                 Bit6 => #emstop,
                 Bit7 => #reserved,
                 Bit8 => #reserved,
                 Bit9 => #reserved,
                 Bit10 => #Pres_low,
                 Bit11 => #reserved,
                 Bit12 => #reserved,
                 Bit13 => #reserved,
                 Bit14 => #reserved,
                 Bit15 => #uti_cv,
                 ENO => #_w1);
   IF #_w1 THEN
       "Bit_to_Word"(Bit0 := #steam_flush,
                     Bit1 := #SUV_flush,
                     Bit2 := #flush_tm_comp,
                     Bit3 := #Vent_tm_comp,
                     Bit4 := #Cond_tm_comp,
                     Bit5 := #reserved,
                     Bit6 := #reserved,
                     Bit7 := #reserved,
                     Bit8 := #reserved,
                     Bit9 := #reserved,
                     Bit10 := #reserved,
                     Bit11 := #reserved,
                     Bit12 := #reserved,
                     Bit13 := #reserved,
                     Bit14 := #reserved,
                     Bit15 := #reserved,
                     "word" => #status);
   END_IF;
END_REGION

REGION Network 6: Brine select
   // Brine select
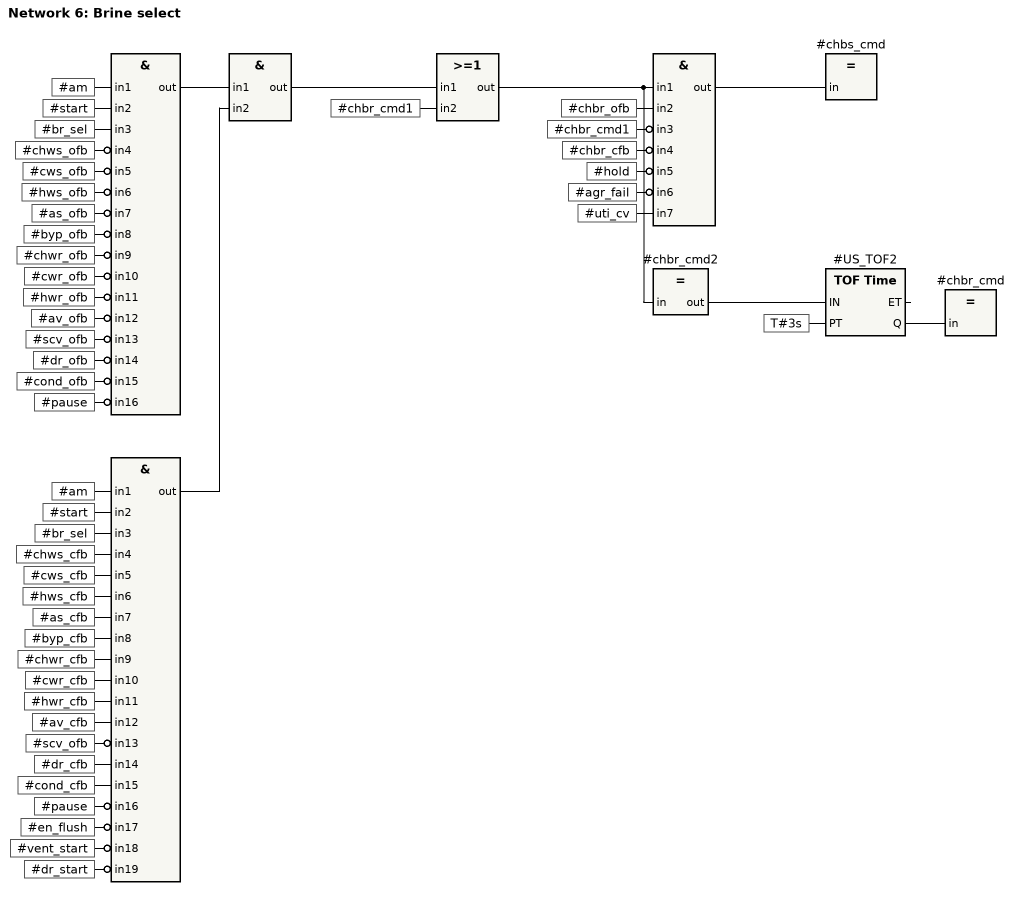
   #_w1 := (#am AND #start AND #br_sel AND NOT #chws_ofb AND NOT #cws_ofb AND NOT #hws_ofb AND NOT #as_ofb AND NOT #byp_ofb AND NOT #chwr_ofb AND NOT #cwr_ofb AND NOT #hwr_ofb AND NOT #av_ofb AND NOT #scv_ofb AND NOT #dr_ofb AND NOT #cond_ofb AND NOT #pause AND #am AND #start AND #br_sel AND #chws_cfb AND #cws_cfb AND #hws_cfb AND #as_cfb AND #byp_cfb AND #chwr_cfb AND #cwr_cfb AND #hwr_cfb AND #av_cfb AND NOT #scv_ofb AND #dr_cfb AND #cond_cfb AND NOT #pause AND NOT #en_flush AND NOT #vent_start AND NOT #dr_start) OR #chbr_cmd1;
   #chbs_cmd := #_w1 AND #chbr_ofb AND NOT #chbr_cmd1 AND NOT #chbr_cfb AND NOT #hold AND NOT #agr_fail AND #uti_cv;
   #chbr_cmd2 := #_w1;
   #US_TOF2(IN := #_w1, PT := T#3s);   // TOF
   #chbr_cmd := #US_TOF2.Q;
END_REGION

REGION Network 7: CMNR logic
   // CMNR logic
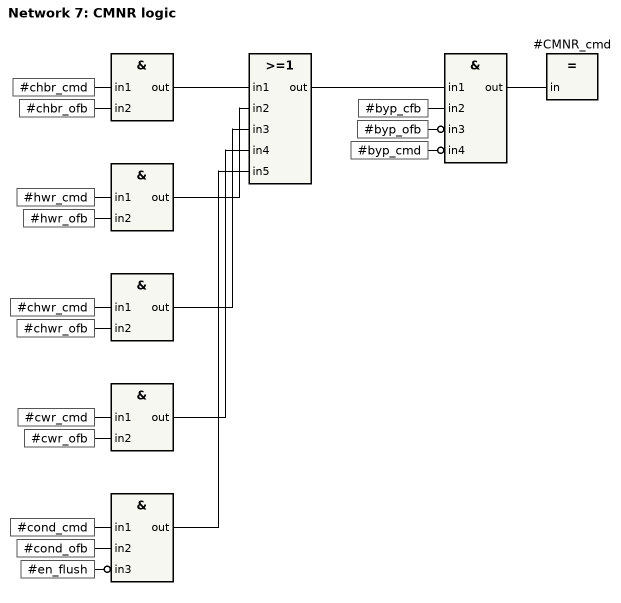
   #CMNR_cmd := ((#chbr_cmd AND #chbr_ofb) OR (#hwr_cmd AND #hwr_ofb) OR (#chwr_cmd AND #chwr_ofb) OR (#cwr_cmd AND #cwr_ofb) OR (#cond_cmd AND #cond_ofb AND NOT #en_flush)) AND #byp_cfb AND NOT #byp_ofb AND NOT #byp_cmd;
END_REGION

REGION Network 8: HW select
   // Hw select
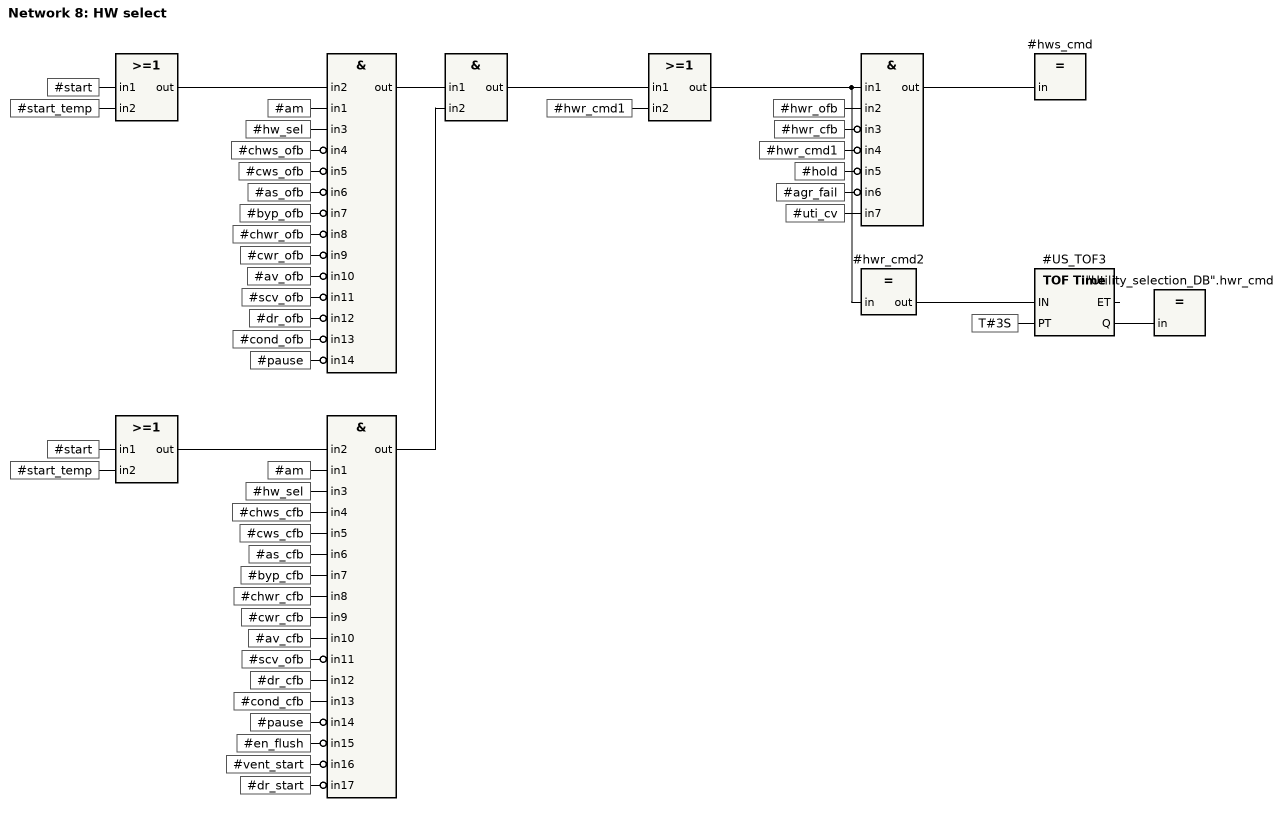
   #_w1 := ((#start OR #start_temp) AND #am AND #hw_sel AND NOT #chws_ofb AND NOT #cws_ofb AND NOT #as_ofb AND NOT #byp_ofb AND NOT #chwr_ofb AND NOT #cwr_ofb AND NOT #av_ofb AND NOT #scv_ofb AND NOT #dr_ofb AND NOT #cond_ofb AND NOT #pause AND (#start OR #start_temp) AND #am AND #hw_sel AND #chws_cfb AND #cws_cfb AND #as_cfb AND #byp_cfb AND #chwr_cfb AND #cwr_cfb AND #av_cfb AND NOT #scv_ofb AND #dr_cfb AND #cond_cfb AND NOT #pause AND NOT #en_flush AND NOT #vent_start AND NOT #dr_start) OR #hwr_cmd1;
   #hws_cmd := #_w1 AND #hwr_ofb AND NOT #hwr_cfb AND NOT #hwr_cmd1 AND NOT #hold AND NOT #agr_fail AND #uti_cv;
   #hwr_cmd2 := #_w1;
   #US_TOF3(IN := #_w1, PT := T#3S);   // TOF
   "Utility_selection_DB".hwr_cmd := #US_TOF3.Q;
END_REGION

REGION Network 9: chw select
   // chw select
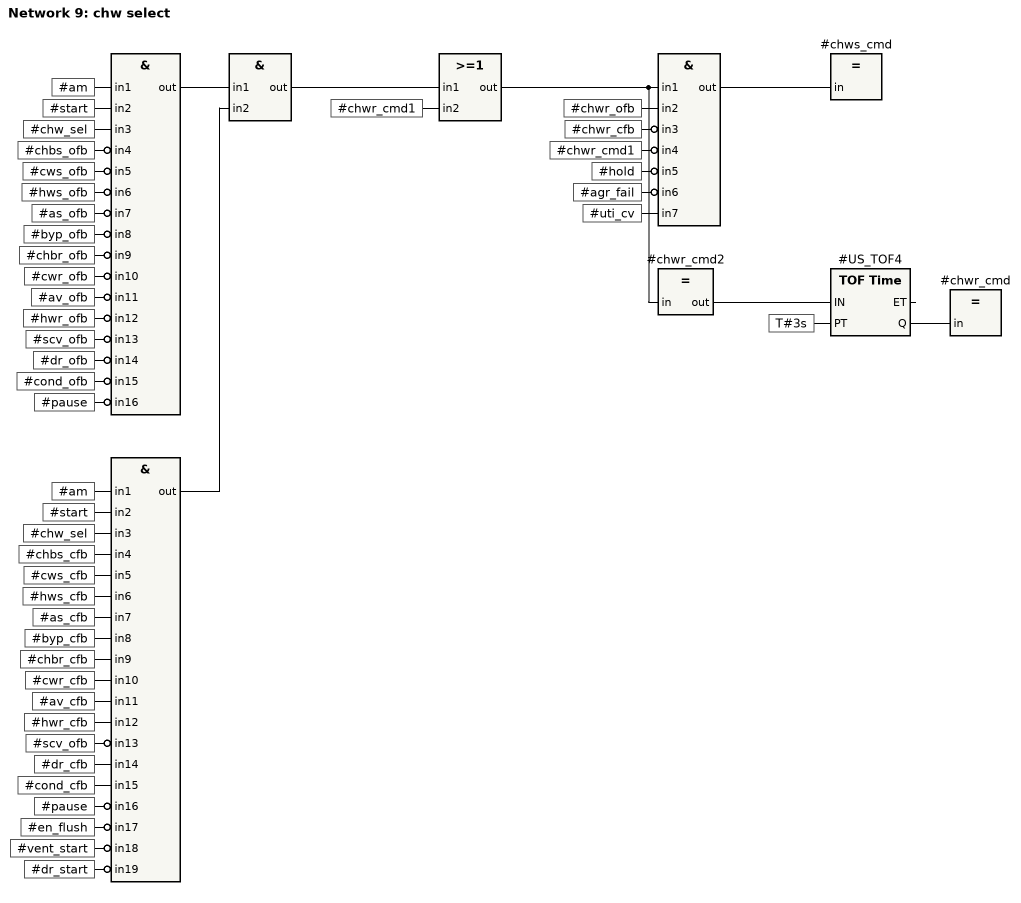
   #_w1 := (#am AND #start AND #chw_sel AND NOT #chbs_ofb AND NOT #cws_ofb AND NOT #hws_ofb AND NOT #as_ofb AND NOT #byp_ofb AND NOT #chbr_ofb AND NOT #cwr_ofb AND NOT #av_ofb AND NOT #hwr_ofb AND NOT #scv_ofb AND NOT #dr_ofb AND NOT #cond_ofb AND NOT #pause AND #am AND #start AND #chw_sel AND #chbs_cfb AND #cws_cfb AND #hws_cfb AND #as_cfb AND #byp_cfb AND #chbr_cfb AND #cwr_cfb AND #av_cfb AND #hwr_cfb AND NOT #scv_ofb AND #dr_cfb AND #cond_cfb AND NOT #pause AND NOT #en_flush AND NOT #vent_start AND NOT #dr_start) OR #chwr_cmd1;
   #chws_cmd := #_w1 AND #chwr_ofb AND NOT #chwr_cfb AND NOT #chwr_cmd1 AND NOT #hold AND NOT #agr_fail AND #uti_cv;
   #chwr_cmd2 := #_w1;
   #US_TOF4(IN := #_w1, PT := T#3s);   // TOF
   #chwr_cmd := #US_TOF4.Q;
END_REGION

REGION Network 10: Steam select
   // Steam select
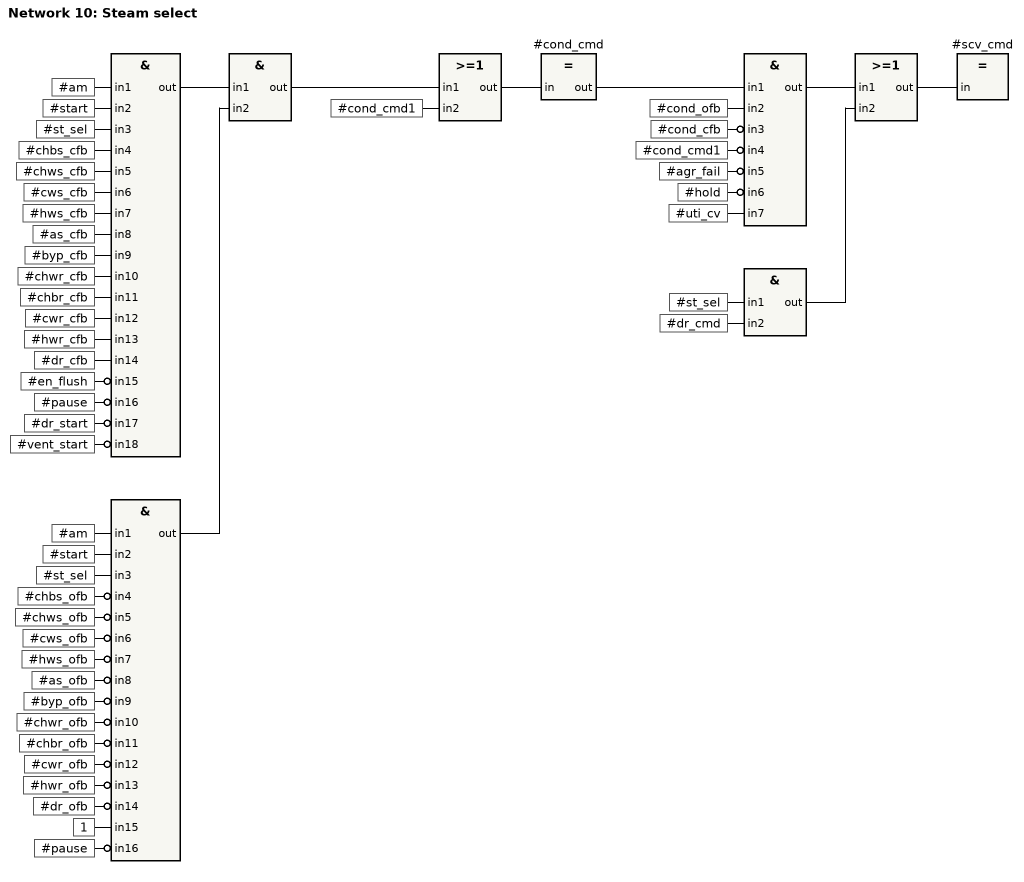
   #cond_cmd := (#am AND #start AND #st_sel AND #chbs_cfb AND #chws_cfb AND #cws_cfb AND #hws_cfb AND #as_cfb AND #byp_cfb AND #chwr_cfb AND #chbr_cfb AND #cwr_cfb AND #hwr_cfb AND #dr_cfb AND NOT #en_flush AND NOT #pause AND NOT #dr_start AND NOT #vent_start AND #am AND #start AND #st_sel AND NOT #chbs_ofb AND NOT #chws_ofb AND NOT #cws_ofb AND NOT #hws_ofb AND NOT #as_ofb AND NOT #byp_ofb AND NOT #chwr_ofb AND NOT #chbr_ofb AND NOT #cwr_ofb AND NOT #hwr_ofb AND NOT #dr_ofb AND 1 AND NOT #pause) OR #cond_cmd1;
   #scv_cmd := (#cond_cmd AND #cond_ofb AND NOT #cond_cfb AND NOT #cond_cmd1 AND NOT #agr_fail AND NOT #hold AND #uti_cv) OR (#st_sel AND #dr_cmd);
END_REGION

REGION Network 11: cw_select
   // cw_select
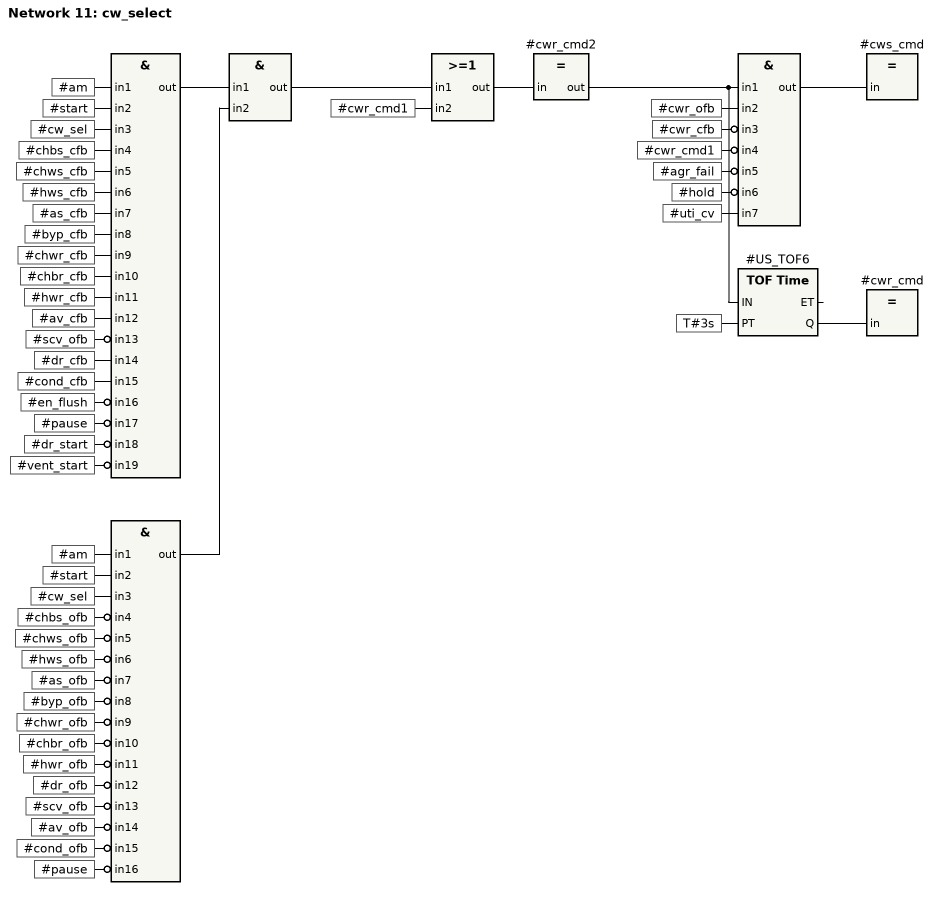
   #cwr_cmd2 := (#am AND #start AND #cw_sel AND #chbs_cfb AND #chws_cfb AND #hws_cfb AND #as_cfb AND #byp_cfb AND #chwr_cfb AND #chbr_cfb AND #hwr_cfb AND #av_cfb AND NOT #scv_ofb AND #dr_cfb AND #cond_cfb AND NOT #en_flush AND NOT #pause AND NOT #dr_start AND NOT #vent_start AND #am AND #start AND #cw_sel AND NOT #chbs_ofb AND NOT #chws_ofb AND NOT #hws_ofb AND NOT #as_ofb AND NOT #byp_ofb AND NOT #chwr_ofb AND NOT #chbr_ofb AND NOT #hwr_ofb AND NOT #dr_ofb AND NOT #scv_ofb AND NOT #av_ofb AND NOT #cond_ofb AND NOT #pause) OR #cwr_cmd1;
   #cws_cmd := #cwr_cmd2 AND #cwr_ofb AND NOT #cwr_cfb AND NOT #cwr_cmd1 AND NOT #agr_fail AND NOT #hold AND #uti_cv;
   #US_TOF6(IN := #cwr_cmd2, PT := T#3s);   // TOF
   #cwr_cmd := #US_TOF6.Q;
END_REGION

REGION Network 12: flush selection
   // flush selection
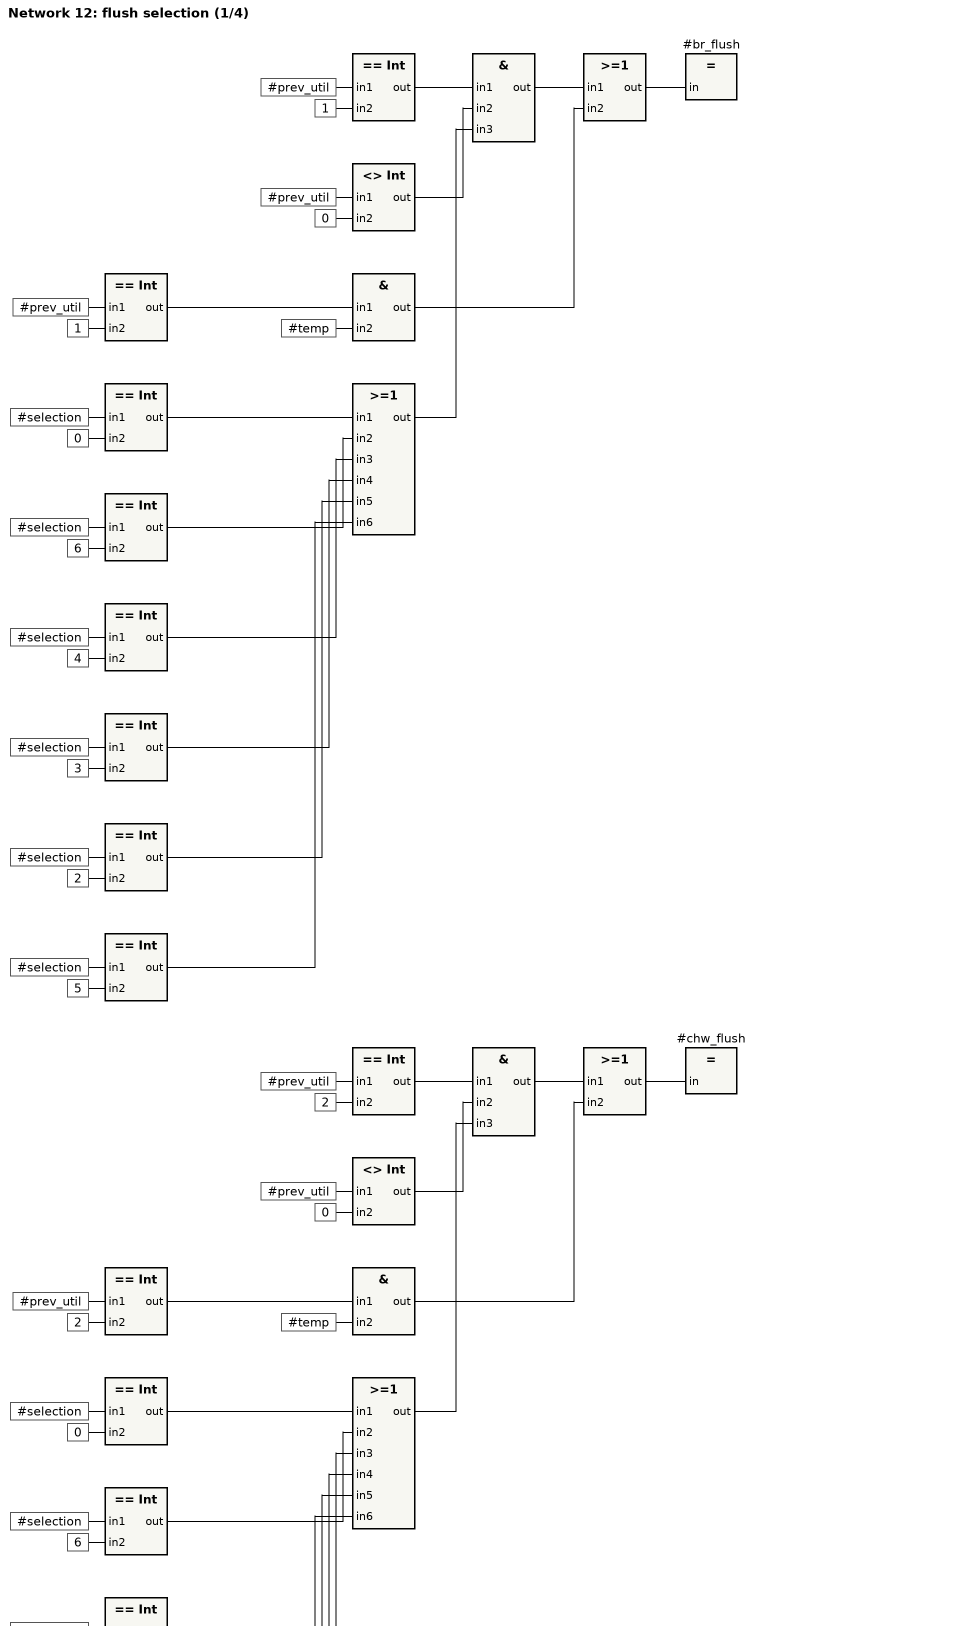
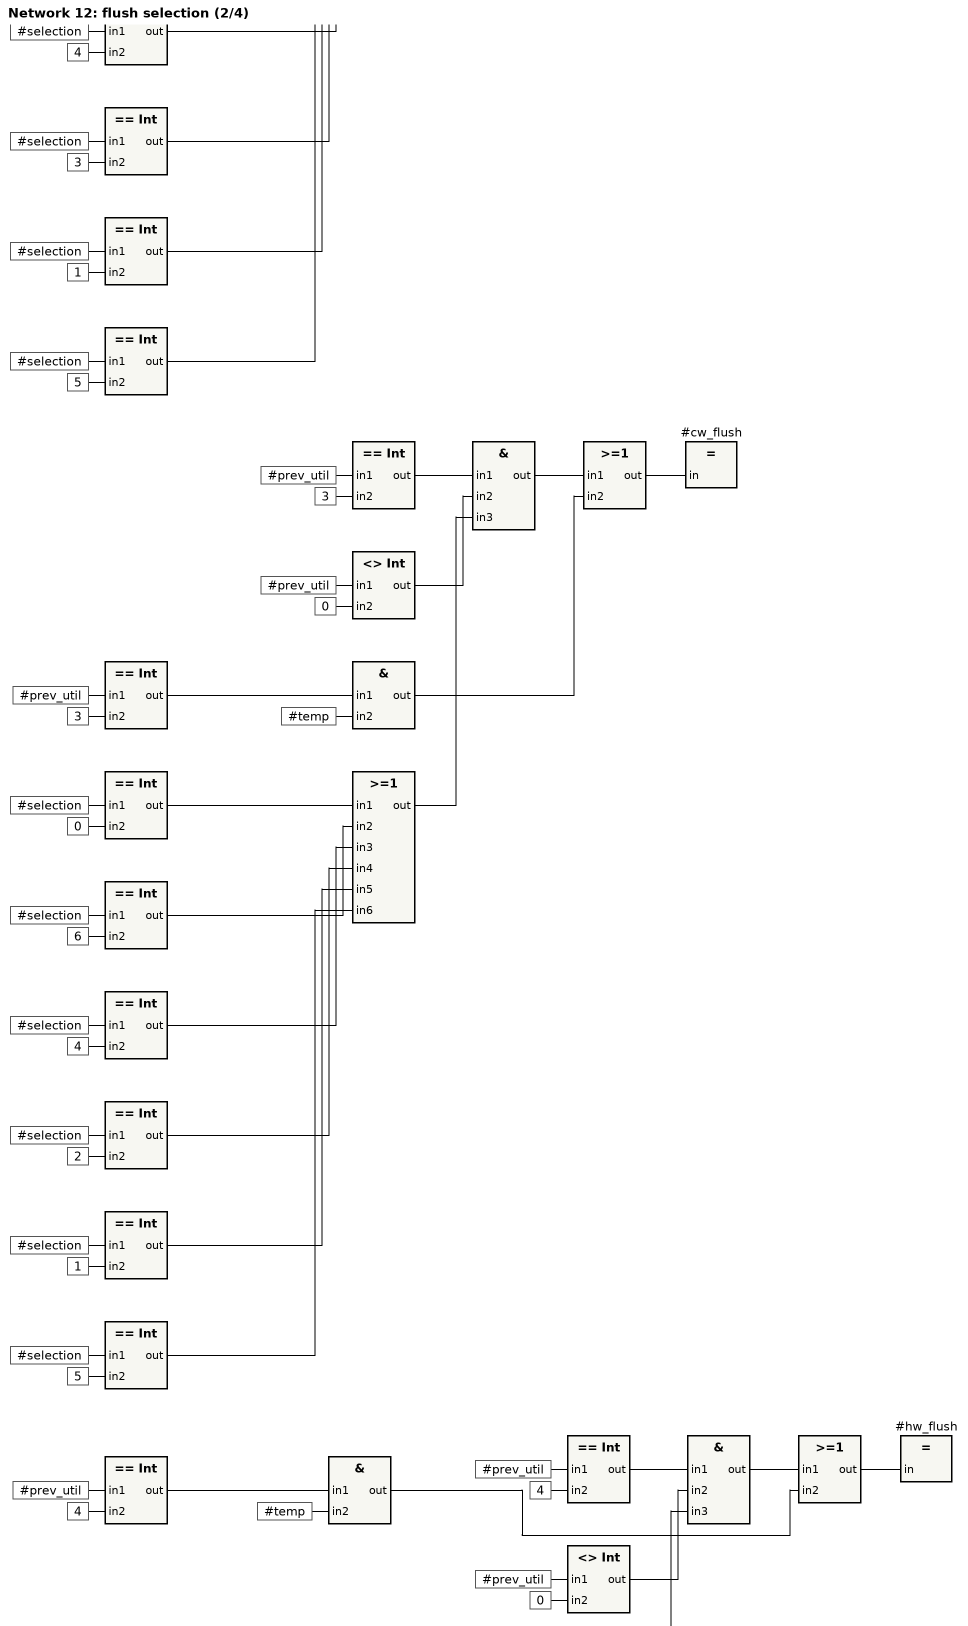
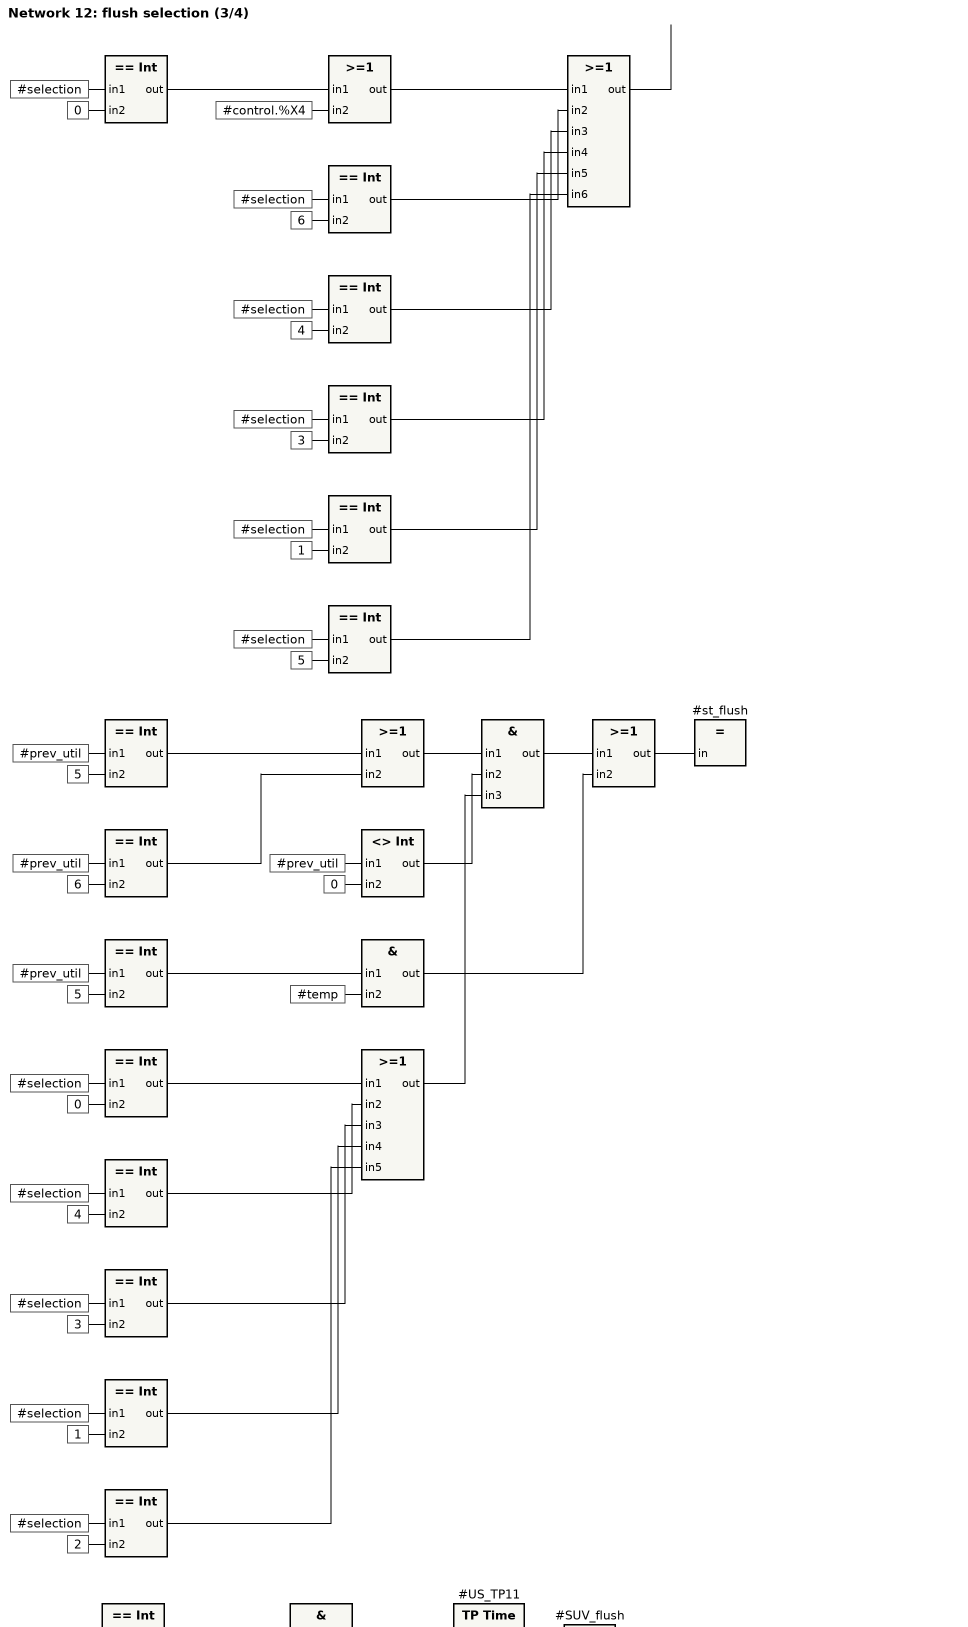
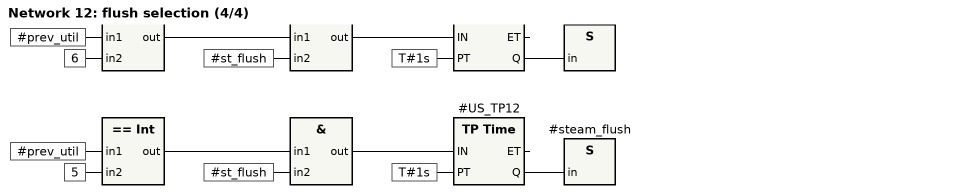
   #br_flush := ((#prev_util = 1) AND (#prev_util <> 0) AND ((#selection = 0) OR (#selection = 6) OR (#selection = 4) OR (#selection = 3) OR (#selection = 2) OR (#selection = 5))) OR ((#prev_util = 1) AND #temp);
   #chw_flush := ((#prev_util = 2) AND (#prev_util <> 0) AND ((#selection = 0) OR (#selection = 6) OR (#selection = 4) OR (#selection = 3) OR (#selection = 1) OR (#selection = 5))) OR ((#prev_util = 2) AND #temp);
   #cw_flush := ((#prev_util = 3) AND (#prev_util <> 0) AND ((#selection = 0) OR (#selection = 6) OR (#selection = 4) OR (#selection = 2) OR (#selection = 1) OR (#selection = 5))) OR ((#prev_util = 3) AND #temp);
   #hw_flush := ((#prev_util = 4) AND (#prev_util <> 0) AND ((#selection = 0) OR #control.%X4 OR (#selection = 6) OR (#selection = 4) OR (#selection = 3) OR (#selection = 1) OR (#selection = 5))) OR ((#prev_util = 4) AND #temp);
   #st_flush := (((#prev_util = 5) OR (#prev_util = 6)) AND (#prev_util <> 0) AND ((#selection = 0) OR (#selection = 4) OR (#selection = 3) OR (#selection = 1) OR (#selection = 2))) OR ((#prev_util = 5) AND #temp);
   #US_TP11(IN := (#prev_util = 6) AND #st_flush, PT := T#1s);   // TP
   IF #US_TP11.Q THEN #SUV_flush := TRUE; END_IF;
   #US_TP12(IN := (#prev_util = 5) AND #st_flush, PT := T#1s);   // TP
   IF #US_TP12.Q THEN #steam_flush := TRUE; END_IF;
END_REGION

REGION Network 13: Flushing Timer
   // Flushing timer
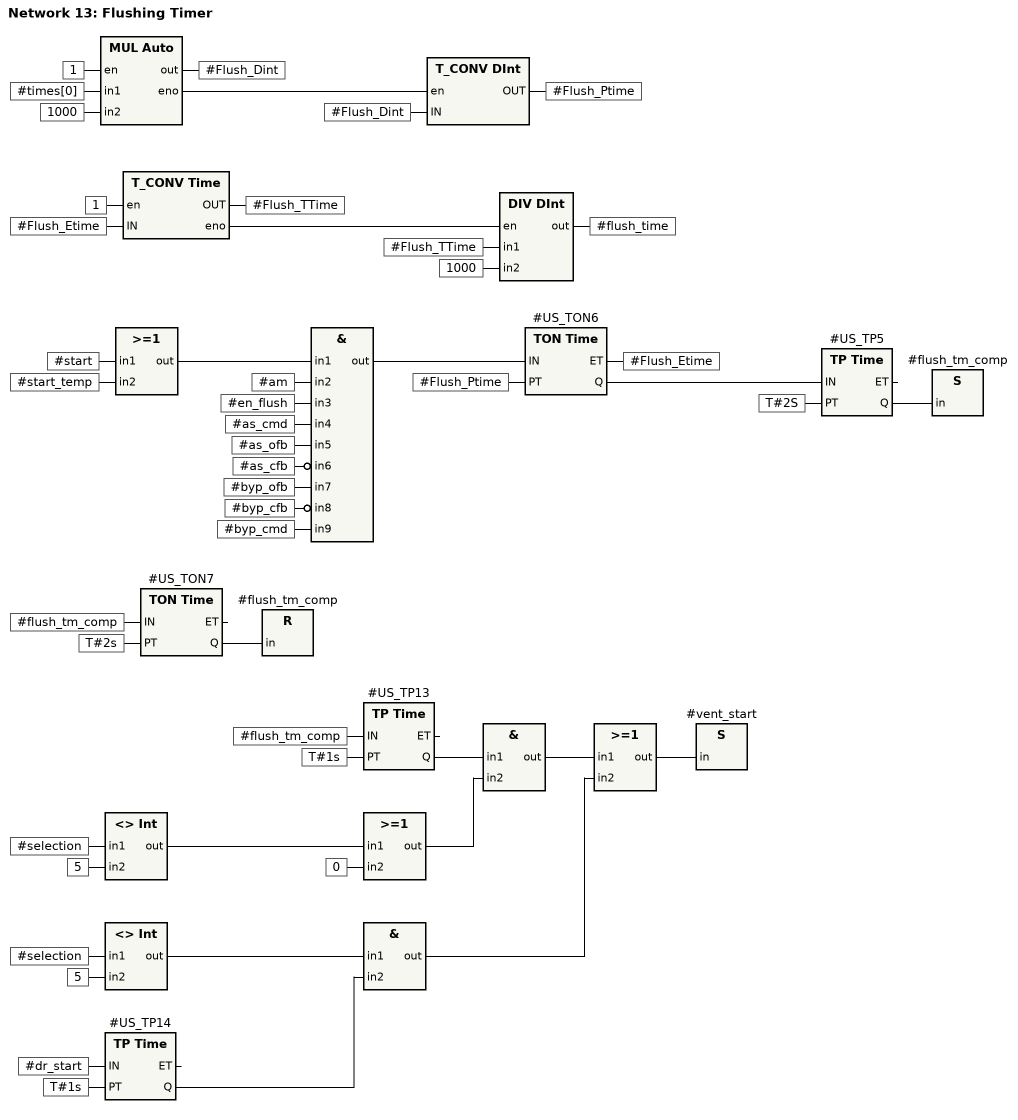
   IF 1 THEN
       #Flush_Dint := #times[0] * 1000;
       T_CONV(IN := #Flush_Dint, OUT => #Flush_Ptime);
   END_IF;
   T_CONV(EN := 1, IN := #Flush_Etime, OUT => #Flush_TTime, ENO => #_w1);
   IF #_w1 THEN #flush_time := #Flush_TTime / 1000; END_IF;
   #US_TON6(IN := (#start OR #start_temp) AND #am AND #en_flush AND #as_cmd AND #as_ofb AND NOT #as_cfb AND #byp_ofb AND NOT #byp_cfb AND #byp_cmd,   // TON
            PT := #Flush_Ptime,
            ET => #Flush_Etime);
   #US_TP5(IN := #US_TON6.Q, PT := T#2S);   // TP
   IF #US_TP5.Q THEN #flush_tm_comp := TRUE; END_IF;
   #US_TON7(IN := #flush_tm_comp, PT := T#2s);   // TON
   IF #US_TON7.Q THEN #flush_tm_comp := FALSE; END_IF;
   #US_TP13(IN := #flush_tm_comp, PT := T#1s);   // TP
   #US_TP14(IN := #dr_start, PT := T#1s);   // TP
   IF (#US_TP13.Q AND ((#selection <> 5) OR 0)) OR ((#selection <> 5) AND #US_TP14.Q) THEN
       #vent_start := TRUE;
   END_IF;
END_REGION

REGION Network 14: vent timer
   // vent timer
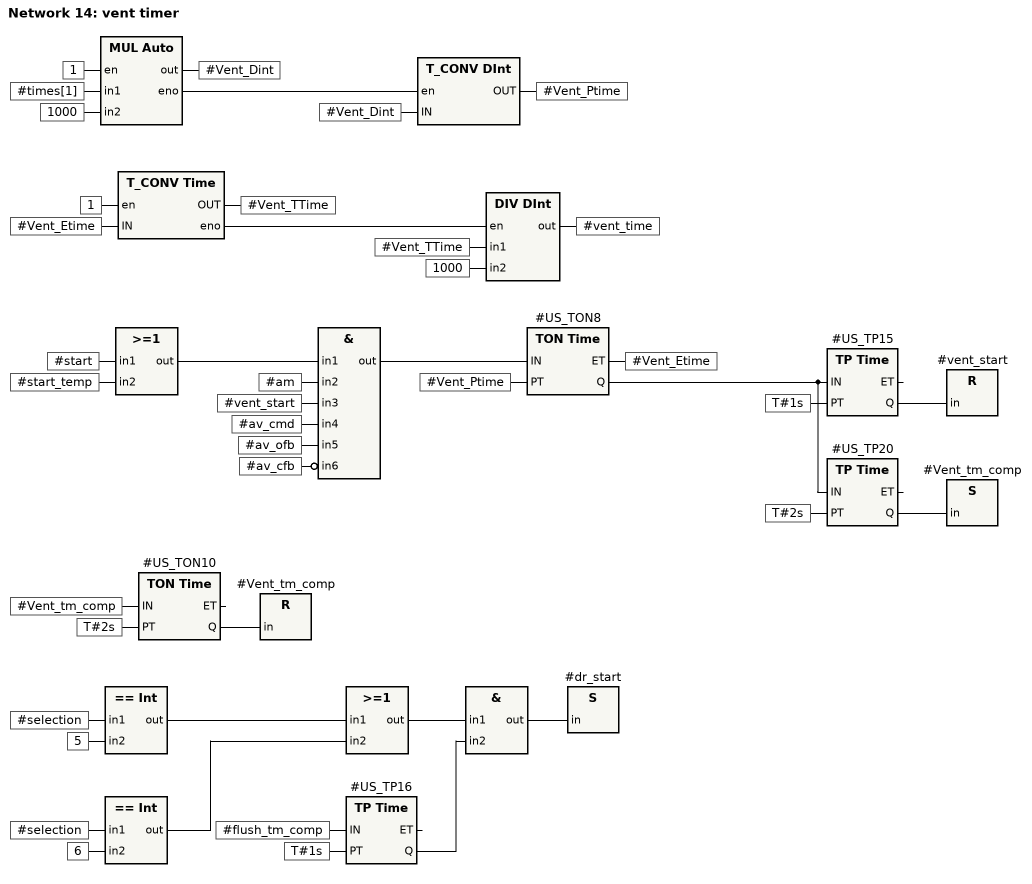
   IF 1 THEN
       #Vent_Dint := #times[1] * 1000;
       T_CONV(IN := #Vent_Dint, OUT => #Vent_Ptime);
   END_IF;
   T_CONV(EN := 1, IN := #Vent_Etime, OUT => #Vent_TTime, ENO => #_w1);
   IF #_w1 THEN #vent_time := #Vent_TTime / 1000; END_IF;
   #US_TON8(IN := (#start OR #start_temp) AND #am AND #vent_start AND #av_cmd AND #av_ofb AND NOT #av_cfb,   // TON
            PT := #Vent_Ptime,
            ET => #Vent_Etime);
   #US_TP15(IN := #US_TON8.Q, PT := T#1s);   // TP
   IF #US_TP15.Q THEN #vent_start := FALSE; END_IF;
   #US_TP20(IN := #US_TON8.Q, PT := T#2s);   // TP
   IF #US_TP20.Q THEN #Vent_tm_comp := TRUE; END_IF;
   #US_TON10(IN := #Vent_tm_comp, PT := T#2s);   // TON
   IF #US_TON10.Q THEN #Vent_tm_comp := FALSE; END_IF;
   #US_TP16(IN := #flush_tm_comp, PT := T#1s);   // TP
   IF ((#selection = 5) OR (#selection = 6)) AND #US_TP16.Q THEN #dr_start := TRUE; END_IF;
END_REGION

REGION Network 15: Condensation timer
   // condensation timer
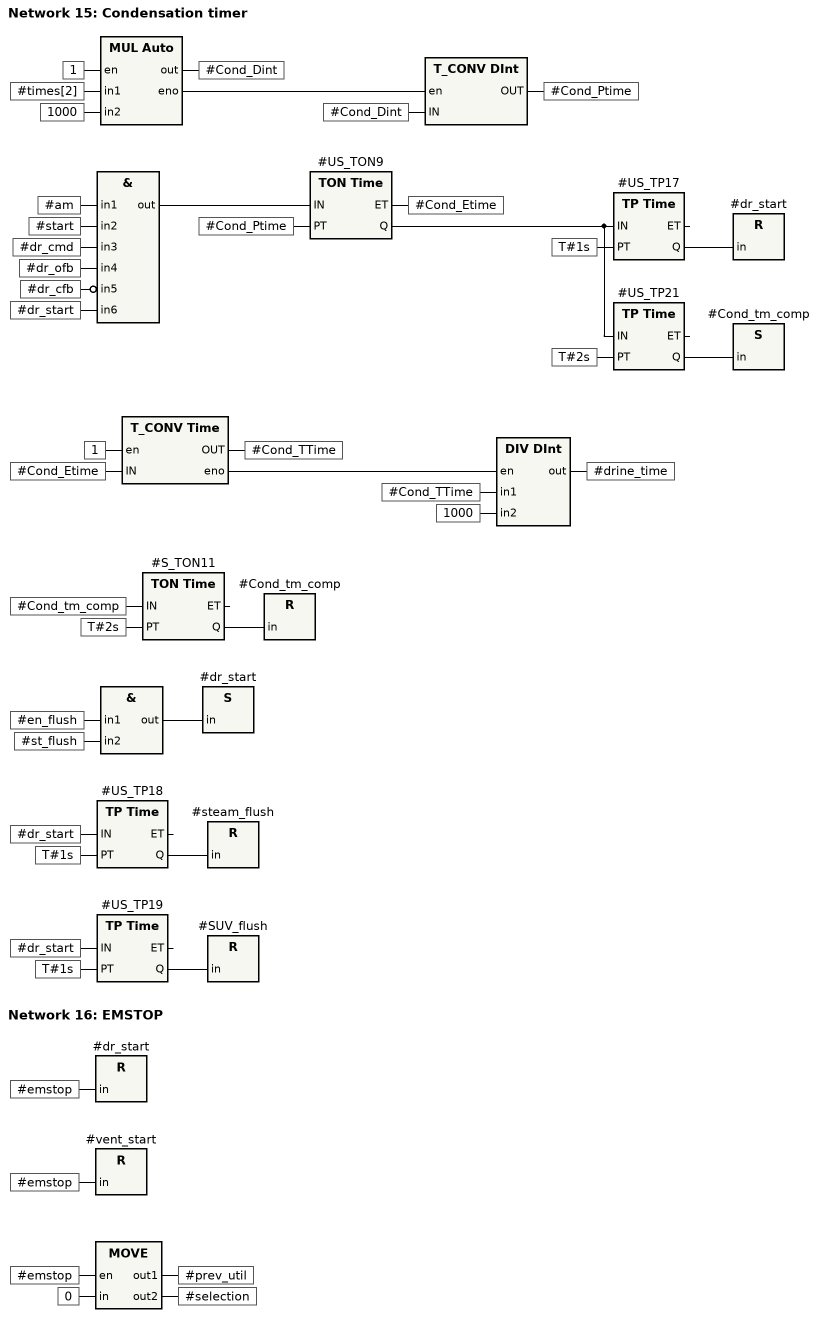
   IF 1 THEN
       #Cond_Dint := #times[2] * 1000;
       T_CONV(IN := #Cond_Dint, OUT => #Cond_Ptime);
   END_IF;
   #US_TON9(IN := #am AND #start AND #dr_cmd AND #dr_ofb AND NOT #dr_cfb AND #dr_start,   // TON
            PT := #Cond_Ptime,
            ET => #Cond_Etime);
   #US_TP17(IN := #US_TON9.Q, PT := T#1s);   // TP
   IF #US_TP17.Q THEN #dr_start := FALSE; END_IF;
   #US_TP21(IN := #US_TON9.Q, PT := T#2s);   // TP
   IF #US_TP21.Q THEN #Cond_tm_comp := TRUE; END_IF;
   T_CONV(EN := 1, IN := #Cond_Etime, OUT => #Cond_TTime, ENO => #_w1);
   IF #_w1 THEN #drine_time := #Cond_TTime / 1000; END_IF;
   #S_TON11(IN := #Cond_tm_comp, PT := T#2s);   // TON
   IF #S_TON11.Q THEN #Cond_tm_comp := FALSE; END_IF;
   IF #en_flush AND #st_flush THEN #dr_start := TRUE; END_IF;
   #US_TP18(IN := #dr_start, PT := T#1s);   // TP
   IF #US_TP18.Q THEN #steam_flush := FALSE; END_IF;
   #US_TP19(IN := #dr_start, PT := T#1s);   // TP
   IF #US_TP19.Q THEN #SUV_flush := FALSE; END_IF;
END_REGION

REGION Network 16: EMSTOP
   // EMSTOP
   IF #emstop THEN
       #dr_start := FALSE;
       #vent_start := FALSE;
       #prev_util := 0;
       #selection := 0;
   END_IF;
END_REGION

REGION Network 17: Brine flushing logic
   // Brine flushing logic
